LIN {X 0,Y 421.138,Z 564.023,A -85,B 0,C 180,E1 -10017.814,E2 -10017.814} C_VEL
LIN {X 0,Y 421.923,Z 552.011,A -85,B 0,C 180,E1 -10018.748,E2 -10018.748} C_VEL
LIN {X 0,Y 422.666,Z 540.319,A -85,B 0,C 180,E1 -10019.442,E2 -10019.442} C_VEL
LIN {X 0,Y 423.16,Z 527.88,A -85,B 0,C 180,E1 -10019.985,E2 -10019.985} C_VEL
LIN {X 0,Y 423.537,Z 514.922,A -85,B 0,C 180,E1 -10020.346,E2 -10020.346} C_VEL
LIN {X 0,Y 424.553,Z 431.561,A -85,B 0,C 180,E1 -10021.795,E2 -10021.795} C_VEL
LIN {X 0,Y 420.563,Z 412.408,A -85,B 0,C 180,E1 -10022.358,E2 -10022.358} C_VEL
LIN {X 0,Y 420.281,Z 410.463,A -85,B 0,C 180,E1 -10022.492,E2 -10022.492} C_VEL
LIN {X 0,Y 420.893,Z 401.257,A -85,B 0,C 180,E1 -10024.591,E2 -10024.591} C_VEL
LIN {X 0,Y 420.17,Z 396.256,A -85,B 0,C 180,E1 -10025.832,E2 -10025.832} C_VEL
LIN {X 0,Y 418.279,Z 386.932,A -85,B 0,C 180,E1 -10028.302,E2 -10028.302} C_VEL
LIN {X 0,Y 418.263,Z 386.884,A -85,B 0,C 180,E1 -10030.942,E2 -10030.942} C_VEL
LIN {X 0,Y 418.279,Z 386.883,A -85,B 0,C 180,E1 -10033.739,E2 -10033.739} C_VEL
LIN {X 0,Y 418.263,Z 386.884,A -85,B 0,C 180,E1 -10036.456,E2 -10036.456} C_VEL
LIN {X 0,Y 418.262,Z 386.885,A -85,B 0,C 180,E1 -10039.122,E2 -10039.122} C_VEL
LIN {X 0,Y 418.233,Z 386.883,A -85,B 0,C 180,E1 -10042.164,E2 -10042.164} C_VEL
LIN {X 0,Y 418.259,Z 386.876,A -85,B 0,C 180,E1 -10045.419,E2 -10045.419} C_VEL
LIN {X 0,Y 418.217,Z 386.89,A -85,B 0,C 180,E1 -10048.604,E2 -10048.604} C_VEL
LIN {X 0,Y 418.288,Z 386.877,A -85,B 0,C 180,E1 -10051.936,E2 -10051.936} C_VEL
LIN {X 0,Y 418.282,Z 386.882,A -85,B 0,C 180,E1 -10055.162,E2 -10055.162} C_VEL
LIN {X 0,Y 418.247,Z 386.88,A -85,B 0,C 180,E1 -10058.304,E2 -10058.304} C_VEL
LIN {X 0,Y 418.276,Z 386.878,A -85,B 0,C 180,E1 -10061.383,E2 -10061.383} C_VEL
LIN {X 0,Y 418.294,Z 386.879,A -85,B 0,C 180,E1 -10064.406,E2 -10064.406} C_VEL
LIN {X 0,Y 418.361,Z 386.871,A -85,B 0,C 180,E1 -10067.386,E2 -10067.386} C_VEL
LIN {X 0,Y 418.352,Z 386.865,A -85,B 0,C 180,E1 -10070.329,E2 -10070.329} C_VEL
LIN {X 0,Y 418.485,Z 386.852,A -85,B 0,C 180,E1 -10073.249,E2 -10073.249} C_VEL
LIN {X 0,Y 418.336,Z 386.875,A -85,B 0,C 180,E1 -10075.182,E2 -10075.182} C_VEL
LIN {X 0,Y 418.538,Z 386.846,A -85,B 0,C 180,E1 -10078.076,E2 -10078.076} C_VEL
LIN {X 0,Y 418.665,Z 386.828,A -85,B 0,C 180,E1 -10080,E2 -10080} C_VEL
LIN {X 0,Y 418.504,Z 386.851,A -85,B 0,C 180,E1 -10082.888,E2 -10082.888} C_VEL
LIN {X 0,Y 418.486,Z 386.859,A -85,B 0,C 180,E1 -10086.751,E2 -10086.751} C_VEL
LIN {X 0,Y 418.352,Z 386.867,A -85,B 0,C 180,E1 -10089.671,E2 -10089.671} C_VEL
LIN {X 0,Y 418.347,Z 386.867,A -85,B 0,C 180,E1 -10093.006,E2 -10093.006} C_VEL
LIN {X 0,Y 418.304,Z 386.88,A -85,B 0,C 180,E1 -10096.736,E2 -10096.736} C_VEL
LIN {X 0,Y 418.263,Z 386.88,A -85,B 0,C 180,E1 -10099.791,E2 -10099.791} C_VEL
LIN {X 0,Y 418.231,Z 386.884,A -85,B 0,C 180,E1 -10102.737,E2 -10102.737} C_VEL
LIN {X 0,Y 418.264,Z 386.88,A -85,B 0,C 180,E1 -10105.905,E2 -10105.905} C_VEL
LIN {X 0,Y 418.258,Z 386.883,A -85,B 0,C 180,E1 -10109.163,E2 -10109.163} C_VEL
LIN {X 0,Y 418.251,Z 386.886,A -85,B 0,C 180,E1 -10112.845,E2 -10112.845} C_VEL
LIN {X 0,Y 418.243,Z 386.888,A -85,B 0,C 180,E1 -10116.24,E2 -10116.24} C_VEL
LIN {X 0,Y 418.261,Z 386.881,A -85,B 0,C 180,E1 -10119.681,E2 -10119.681} C_VEL
LIN {X 0,Y 418.28,Z 386.87,A -85,B 0,C 180,E1 -10122.33,E2 -10122.33} C_VEL
LIN {X 0,Y 418.251,Z 386.88,A -85,B 0,C 180,E1 -10125.112,E2 -10125.112} C_VEL
LIN {X 0,Y 418.239,Z 386.884,A -85,B 0,C 180,E1 -10127.768,E2 -10127.768} C_VEL
LIN {X 0,Y 418.254,Z 386.881,A -85,B 0,C 180,E1 -10130.619,E2 -10130.619} C_VEL
LIN {X 0,Y 418.244,Z 386.881,A -85,B 0,C 180,E1 -10133.977,E2 -10133.977} C_VEL
LIN {X 0,Y 418.256,Z 386.886,A -85,B 0,C 180,E1 -10137.157,E2 -10137.157} C_VEL
LIN {X 0,Y 418.268,Z 386.886,A -85,B 0,C 180,E1 -10140.896,E2 -10140.896} C_VEL
LIN {X 0,Y 418.343,Z 386.992,A -85,B 0,C 180,E1 -10142.829,E2 -10142.829} C_VEL
LIN {X 0,Y 420.436,Z 396.948,A -85,B 0,C 180,E1 -10145.299,E2 -10145.299} C_VEL
LIN {X 0,Y 421.424,Z 403.012,A -85,B 0,C 180,E1 -10146.715,E2 -10146.715} C_VEL
LIN {X 0,Y 420.312,Z 418.167,A -85,B 0,C 180,E1 -10149.954,E2 -10149.954} C_VEL
LIN {X 0,Y 420.149,Z 421.353,A -85,B 0,C 180,E1 -10150.594,E2 -10150.594} C_VEL
LIN {X 0,Y 421.621,Z 428.874,A -85,B 0,C 180,E1 -10150.85,E2 -10150.85} C_VEL
LIN {X 0,Y 424.489,Z 445.436,A -85,B 0,C 180,E1 -10151.3,E2 -10151.3} C_VEL
LIN {X 0,Y 423.431,Z 529.437,A -85,B 0,C 180,E1 -10152.773,E2 -10152.773} C_VEL
LIN {X 0,Y 422.94,Z 543.257,A -85,B 0,C 180,E1 -10153.219,E2 -10153.219} C_VEL
LIN {X 0,Y 422.283,Z 555.661,A -85,B 0,C 180,E1 -10153.814,E2 -10153.814} C_VEL
LIN {X 0,Y 421.5,Z 566.743,A -85,B 0,C 180,E1 -10154.528,E2 -10154.528} C_VEL
LIN {X 0,Y 420.716,Z 578.277,A -85,B 0,C 180,E1 -10155.489,E2 -10155.489} C_VEL
LIN {X 0,Y 419.929,Z 588.676,A -85,B 0,C 180,E1 -10156.573,E2 -10156.573} C_VEL
LIN {X 0,Y 419.309,Z 597.186,A -85,B 0,C 180,E1 -10157.661,E2 -10157.661} C_VEL
LIN {X 0,Y 418.575,Z 605.051,A -85,B 0,C 180,E1 -10158.867,E2 -10158.867} C_VEL
LIN {X 0,Y 418.026,Z 612.748,A -85,B 0,C 180,E1 -10160.322,E2 -10160.322} C_VEL
LIN {X 0,Y 417.549,Z 618.934,A -85,B 0,C 180,E1 -10161.775,E2 -10161.775} C_VEL
LIN {X 0,Y 417.27,Z 623.86,A -85,B 0,C 180,E1 -10163.229,E2 -10163.229} C_VEL
LIN {X 0,Y 417.161,Z 627.67,A -85,B 0,C 180,E1 -10164.684,E2 -10164.684} C_VEL
LIN {X 0,Y 417.001,Z 630.466,A -85,B 0,C 180,E1 -10166.135,E2 -10166.135} C_VEL
LIN {X 0,Y 417.03,Z 632.726,A -85,B 0,C 180,E1 -10168.069,E2 -10168.069} C_VEL
LIN {X 0,Y 416.992,Z 633.268,A -85,B 0,C 180,E1 -10169.035,E2 -10169.035} C_VEL
LIN {X 0,Y 416.982,Z 633.379,A -85,B 0,C 180,E1 -10170,E2 -10170} C_VEL
LIN {X 0,Y 417.03,Z 632.435,A -85,B 0,C 180,E1 -10171.932,E2 -10171.932} C_VEL
LIN {X 0,Y 416.984,Z 631.378,A -85,B 0,C 180,E1 -10172.898,E2 -10172.898} C_VEL
LIN {X 0,Y 417,Z 629.867,A -85,B 0,C 180,E1 -10173.866,E2 -10173.866} C_VEL
LIN {X 0,Y 417.141,Z 626.813,A -85,B 0,C 180,E1 -10175.317,E2 -10175.317} C_VEL
LIN {X 0,Y 417.244,Z 622.691,A -85,B 0,C 180,E1 -10176.771,E2 -10176.771} C_VEL
LIN {X 0,Y 417.566,Z 616.376,A -85,B 0,C 180,E1 -10178.469,E2 -10178.469} C_VEL
LIN {X 0,Y 417.985,Z 609.49,A -85,B 0,C 180,E1 -10179.924,E2 -10179.924} C_VEL
LIN {X 0,Y 418.42,Z 602.45,A -85,B 0,C 180,E1 -10181.137,E2 -10181.137} C_VEL
LIN {X 0,Y 419.055,Z 593.964,A -85,B 0,C 180,E1 -10182.347,E2 -10182.347} C_VEL
LIN {X 0,Y 419.747,Z 583.455,A -85,B 0,C 180,E1 -10183.557,E2 -10183.557} C_VEL
LIN {X 0,Y 420.461,Z 571.606,A -85,B 0,C 180,E1 -10184.644,E2 -10184.644} C_VEL
LIN {X 0,Y 421.178,Z 559.68,A -85,B 0,C 180,E1 -10185.485,E2 -10185.485} C_VEL
LIN {X 0,Y 421.793,Z 547.253,A -85,B 0,C 180,E1 -10186.144,E2 -10186.144} C_VEL
LIN {X 0,Y 422.289,Z 534.454,A -85,B 0,C 180,E1 -10186.621,E2 -10186.621} C_VEL
LIN {X 0,Y 422.514,Z 520.889,A -85,B 0,C 180,E1 -10186.923,E2 -10186.923} C_VEL
LIN {X 0,Y 423.276,Z 444.977,A -85,B 0,C 180,E1 -10188.213,E2 -10188.213} C_VEL
LIN {X 0,Y 419.583,Z 421.755,A -85,B 0,C 180,E1 -10188.779,E2 -10188.779} C_VEL
LIN {X 0,Y 419.773,Z 417.624,A -85,B 0,C 180,E1 -10189.563,E2 -10189.563} C_VEL
LIN {X 0,Y 420.813,Z 401.434,A -85,B 0,C 180,E1 -10192.923,E2 -10192.923} C_VEL
LIN {X 0,Y 419.777,Z 394.378,A -85,B 0,C 180,E1 -10194.479,E2 -10194.479} C_VEL
LIN {X 0,Y 418.35,Z 386.974,A -85,B 0,C 180,E1 -10196.2,E2 -10196.2} C_VEL
LIN {X 0,Y 418.266,Z 386.886,A -85,B 0,C 180,E1 -10199.161,E2 -10199.161} C_VEL
LIN {X 0,Y 418.258,Z 386.882,A -85,B 0,C 180,E1 -10202.844,E2 -10202.844} C_VEL
LIN {X 0,Y 418.249,Z 386.884,A -85,B 0,C 180,E1 -10206.238,E2 -10206.238} C_VEL
LIN {X 0,Y 418.255,Z 386.886,A -85,B 0,C 180,E1 -10209.681,E2 -10209.681} C_VEL
LIN {X 0,Y 418.231,Z 386.886,A -85,B 0,C 180,E1 -10212.321,E2 -10212.321} C_VEL
LIN {X 0,Y 418.26,Z 386.885,A -85,B 0,C 180,E1 -10215.112,E2 -10215.112} C_VEL
LIN {X 0,Y 418.291,Z 386.881,A -85,B 0,C 180,E1 -10217.773,E2 -10217.773} C_VEL
LIN {X 0,Y 418.264,Z 386.885,A -85,B 0,C 180,E1 -10221.559,E2 -10221.559} C_VEL
LIN {X 0,Y 418.256,Z 386.887,A -85,B 0,C 180,E1 -10225.159,E2 -10225.159} C_VEL
LIN {X 0,Y 418.242,Z 386.888,A -85,B 0,C 180,E1 -10227.471,E2 -10227.471} C_VEL
LIN {X 0,Y 418.265,Z 386.884,A -85,B 0,C 180,E1 -10230.895,E2 -10230.895} C_VEL
LIN {X 0,Y 418.267,Z 386.883,A -85,B 0,C 180,E1 -10234.096,E2 -10234.096} C_VEL
LIN {X 0,Y 418.227,Z 386.891,A -85,B 0,C 180,E1 -10237.263,E2 -10237.263} C_VEL
LIN {X 0,Y 418.278,Z 386.88,A -85,B 0,C 180,E1 -10240.364,E2 -10240.364} C_VEL
LIN {X 0,Y 418.312,Z 386.879,A -85,B 0,C 180,E1 -10243.404,E2 -10243.404} C_VEL
LIN {X 0,Y 418.341,Z 386.876,A -85,B 0,C 180,E1 -10246.999,E2 -10246.999} C_VEL
LIN {X 0,Y 418.335,Z 386.874,A -85,B 0,C 180,E1 -10250.328,E2 -10250.328} C_VEL
LIN {X 0,Y 418.487,Z 386.858,A -85,B 0,C 180,E1 -10253.249,E2 -10253.249} C_VEL
LIN {X 0,Y 418.335,Z 386.877,A -85,B 0,C 180,E1 -10255.181,E2 -10255.181} C_VEL
LIN {X 0,Y 418.539,Z 386.849,A -85,B 0,C 180,E1 -10258.075,E2 -10258.075} C_VEL
LIN {X 0,Y 418.666,Z 386.833,A -85,B 0,C 180,E1 -10260,E2 -10260} C_VEL
LIN {X 0,Y 418.505,Z 386.855,A -85,B 0,C 180,E1 -10262.888,E2 -10262.888} C_VEL
LIN {X 0,Y 418.488,Z 386.857,A -85,B 0,C 180,E1 -10266.751,E2 -10266.751} C_VEL
LIN {X 0,Y 418.335,Z 386.876,A -85,B 0,C 180,E1 -10269.671,E2 -10269.671} C_VEL
LIN {X 0,Y 418.34,Z 386.876,A -85,B 0,C 180,E1 -10273.001,E2 -10273.001} C_VEL
LIN {X 0,Y 418.307,Z 386.879,A -85,B 0,C 180,E1 -10276.736,E2 -10276.736} C_VEL
LIN {X 0,Y 418.265,Z 386.884,A -85,B 0,C 180,E1 -10279.79,E2 -10279.79} C_VEL
LIN {X 0,Y 418.233,Z 386.889,A -85,B 0,C 180,E1 -10282.736,E2 -10282.736} C_VEL
LIN {X 0,Y 418.266,Z 386.883,A -85,B 0,C 180,E1 -10285.904,E2 -10285.904} C_VEL
LIN {X 0,Y 418.27,Z 386.884,A -85,B 0,C 180,E1 -10289.162,E2 -10289.162} C_VEL
LIN {X 0,Y 418.254,Z 386.886,A -85,B 0,C 180,E1 -10292.844,E2 -10292.844} C_VEL
LIN {X 0,Y 418.245,Z 386.885,A -85,B 0,C 180,E1 -10296.239,E2 -10296.239} C_VEL
LIN {X 0,Y 418.249,Z 386.885,A -85,B 0,C 180,E1 -10299.682,E2 -10299.682} C_VEL
LIN {X 0,Y 418.229,Z 386.887,A -85,B 0,C 180,E1 -10302.322,E2 -10302.322} C_VEL
LIN {X 0,Y 418.235,Z 386.89,A -85,B 0,C 180,E1 -10305.109,E2 -10305.109} C_VEL
LIN {X 0,Y 418.254,Z 386.884,A -85,B 0,C 180,E1 -10307.769,E2 -10307.769} C_VEL
LIN {X 0,Y 418.266,Z 386.883,A -85,B 0,C 180,E1 -10310.617,E2 -10310.617} C_VEL
LIN {X 0,Y 418.245,Z 386.884,A -85,B 0,C 180,E1 -10313.977,E2 -10313.977} C_VEL
LIN {X 0,Y 418.257,Z 386.888,A -85,B 0,C 180,E1 -10317.156,E2 -10317.156} C_VEL
LIN {X 0,Y 418.268,Z 386.885,A -85,B 0,C 180,E1 -10320.896,E2 -10320.896} C_VEL
LIN {X 0,Y 418.271,Z 386.88,A -85,B 0,C 180,E1 -10324.096,E2 -10324.096} C_VEL
LIN {X 0,Y 418.239,Z 386.888,A -85,B 0,C 180,E1 -10327.264,E2 -10327.264} C_VEL
LIN {X 0,Y 418.284,Z 386.879,A -85,B 0,C 180,E1 -10330.364,E2 -10330.364} C_VEL
LIN {X 0,Y 418.318,Z 386.876,A -85,B 0,C 180,E1 -10333.405,E2 -10333.405} C_VEL
LIN {X 0,Y 418.348,Z 386.877,A -85,B 0,C 180,E1 -10336.999,E2 -10336.999} C_VEL
LIN {X 0,Y 418.318,Z 386.913,A -85,B 0,C 180,E1 -10338.737,E2 -10338.737} C_VEL
LIN {X 0,Y 419.362,Z 392.298,A -85,B 0,C 180,E1 -10340.109,E2 -10340.109} C_VEL
LIN {X 0,Y 420.285,Z 398.53,A -85,B 0,C 180,E1 -10341.586,E2 -10341.586} C_VEL
LIN {X 0,Y 419.795,Z 404.966,A -85,B 0,C 180,E1 -10343.028,E2 -10343.028} C_VEL
LIN {X 0,Y 419.5,Z 409.848,A -85,B 0,C 180,E1 -10344.11,E2 -10344.11} C_VEL
LIN {X 0,Y 419.508,Z 410.969,A -85,B 0,C 180,E1 -10344.274,E2 -10344.274} C_VEL
LIN {X 0,Y 422.211,Z 425.053,A -85,B 0,C 180,E1 -10344.648,E2 -10344.648} C_VEL
LIN {X 0,Y 423.411,Z 432.135,A -85,B 0,C 180,E1 -10344.818,E2 -10344.818} C_VEL
LIN {X 0,Y 422.442,Z 518.153,A -85,B 0,C 180,E1 -10346.304,E2 -10346.304} C_VEL
LIN {X 0,Y 422.1,Z 529.926,A -85,B 0,C 180,E1 -10346.669,E2 -10346.669} C_VEL
LIN {X 0,Y 420.303,Z 537.386,A -85,B 0,C 180,E1 -10346.935,E2 -10346.935} C_VEL
LIN {X 0,Y 417.529,Z 544.56,A -85,B 0,C 180,E1 -10347.223,E2 -10347.223} C_VEL
LIN {X 0,Y 414.552,Z 553.329,A -85,B 0,C 180,E1 -10347.702,E2 -10347.702} C_VEL
LIN {X 0,Y 413.762,Z 558.483,A -85,B 0,C 180,E1 -10348.072,E2 -10348.072} C_VEL
LIN {X 0,Y 413.074,Z 569.244,A -85,B 0,C 180,E1 -10349.025,E2 -10349.025} C_VEL
LIN {X 0,Y 412.365,Z 578.193,A -85,B 0,C 180,E1 -10350,E2 -10350} C_VEL
LIN {X 0,Y 411.779,Z 587.346,A -85,B 0,C 180,E1 -10351.222,E2 -10351.222} C_VEL
LIN {X 0,Y 411.1,Z 596.284,A -85,B 0,C 180,E1 -10352.694,E2 -10352.694} C_VEL
LIN {X 0,Y 410.64,Z 603.483,A -85,B 0,C 180,E1 -10354.171,E2 -10354.171} C_VEL
LIN {X 0,Y 410.383,Z 608.342,A -85,B 0,C 180,E1 -10355.404,E2 -10355.404} C_VEL
LIN {X 0,Y 410.176,Z 613.073,A -85,B 0,C 180,E1 -10356.888,E2 -10356.888} C_VEL
LIN {X 0,Y 409.998,Z 616.699,A -85,B 0,C 180,E1 -10358.378,E2 -10358.378} C_VEL
LIN {X 0,Y 409.821,Z 619.308,A -85,B 0,C 180,E1 -10359.874,E2 -10359.874} C_VEL
LIN {X 0,Y 409.852,Z 620.528,A -85,B 0,C 180,E1 -10360.872,E2 -10360.872} C_VEL
LIN {X 0,Y 409.883,Z 621.466,A -85,B 0,C 180,E1 -10362.22,E2 -10362.22} C_VEL
LIN {X 0,Y 409.755,Z 621.629,A -85,B 0,C 180,E1 -10363.893,E2 -10363.893} C_VEL
LIN {X 0,Y 409.778,Z 621.181,A -85,B 0,C 180,E1 -10364.907,E2 -10364.907} C_VEL
LIN {X 0,Y 409.86,Z 619.948,A -85,B 0,C 180,E1 -10366.209,E2 -10366.209} C_VEL
LIN {X 0,Y 410.018,Z 617.188,A -85,B 0,C 180,E1 -10367.97,E2 -10367.97} C_VEL
LIN {X 0,Y 410.269,Z 613.417,A -85,B 0,C 180,E1 -10369.582,E2 -10369.582} C_VEL
LIN {X 0,Y 410.586,Z 608.813,A -85,B 0,C 180,E1 -10371.066,E2 -10371.066} C_VEL
LIN {X 0,Y 411.167,Z 601.801,A -85,B 0,C 180,E1 -10372.81,E2 -10372.81} C_VEL
LIN {X 0,Y 411.73,Z 594.877,A -85,B 0,C 180,E1 -10374.183,E2 -10374.183} C_VEL
LIN {X 0,Y 412.462,Z 586.649,A -85,B 0,C 180,E1 -10375.516,E2 -10375.516} C_VEL
LIN {X 0,Y 413.27,Z 576.951,A -85,B 0,C 180,E1 -10376.785,E2 -10376.785} C_VEL
LIN {X 0,Y 414.145,Z 566.829,A -85,B 0,C 180,E1 -10377.854,E2 -10377.854} C_VEL
LIN {X 0,Y 414.981,Z 554.936,A -85,B 0,C 180,E1 -10378.859,E2 -10378.859} C_VEL
LIN {X 0,Y 415.794,Z 542.865,A -85,B 0,C 180,E1 -10379.629,E2 -10379.629} C_VEL
LIN {X 0,Y 416.433,Z 529.777,A -85,B 0,C 180,E1 -10380.242,E2 -10380.242} C_VEL
LIN {X 0,Y 416.877,Z 517.663,A -85,B 0,C 180,E1 -10380.618,E2 -10380.618} C_VEL
LIN {X 0,Y 417.981,Z 432.664,A -85,B 0,C 180,E1 -10382.127,E2 -10382.127} C_VEL
LIN {X 0,Y 413.773,Z 412.697,A -85,B 0,C 180,E1 -10382.735,E2 -10382.735} C_VEL
LIN {X 0,Y 413.455,Z 410.579,A -85,B 0,C 180,E1 -10382.875,E2 -10382.875} C_VEL
LIN {X 0,Y 413.984,Z 402.873,A -85,B 0,C 180,E1 -10384.659,E2 -10384.659} C_VEL
LIN {X 0,Y 413.541,Z 399.14,A -85,B 0,C 180,E1 -10385.594,E2 -10385.594} C_VEL
LIN {X 0,Y 411.249,Z 387.872,A -85,B 0,C 180,E1 -10388.594,E2 -10388.594} C_VEL
LIN {X 0,Y 411.217,Z 387.764,A -85,B 0,C 180,E1 -10391.799,E2 -10391.799} C_VEL
LIN {X 0,Y 411.232,Z 387.761,A -85,B 0,C 180,E1 -10394.481,E2 -10394.481} C_VEL
LIN {X 0,Y 411.224,Z 387.758,A -85,B 0,C 180,E1 -10397.296,E2 -10397.296} C_VEL
LIN {X 0,Y 411.226,Z 387.757,A -85,B 0,C 180,E1 -10400.777,E2 -10400.777} C_VEL
LIN {X 0,Y 411.194,Z 387.762,A -85,B 0,C 180,E1 -10404.471,E2 -10404.471} C_VEL
LIN {X 0,Y 411.166,Z 387.766,A -85,B 0,C 180,E1 -10408.003,E2 -10408.003} C_VEL
LIN {X 0,Y 411.217,Z 387.757,A -85,B 0,C 180,E1 -10411.41,E2 -10411.41} C_VEL
LIN {X 0,Y 411.229,Z 387.759,A -85,B 0,C 180,E1 -10414.706,E2 -10414.706} C_VEL
LIN {X 0,Y 411.222,Z 387.754,A -85,B 0,C 180,E1 -10417.914,E2 -10417.914} C_VEL
LIN {X 0,Y 411.228,Z 387.758,A -85,B 0,C 180,E1 -10421.052,E2 -10421.052} C_VEL
LIN {X 0,Y 411.246,Z 387.756,A -85,B 0,C 180,E1 -10424.131,E2 -10424.131} C_VEL
LIN {X 0,Y 411.306,Z 387.752,A -85,B 0,C 180,E1 -10427.166,E2 -10427.166} C_VEL
LIN {X 0,Y 411.3,Z 387.742,A -85,B 0,C 180,E1 -10430.161,E2 -10430.161} C_VEL
LIN {X 0,Y 411.452,Z 387.729,A -85,B 0,C 180,E1 -10433.133,E2 -10433.133} C_VEL
LIN {X 0,Y 411.307,Z 387.749,A -85,B 0,C 180,E1 -10435.099,E2 -10435.099} C_VEL
LIN {X 0,Y 411.507,Z 387.721,A -85,B 0,C 180,E1 -10438.043,E2 -10438.043} C_VEL
LIN {X 0,Y 411.635,Z 387.703,A -85,B 0,C 180,E1 -10440,E2 -10440} C_VEL
LIN {X 0,Y 411.459,Z 387.727,A -85,B 0,C 180,E1 -10442.937,E2 -10442.937} C_VEL
LIN {X 0,Y 411.452,Z 387.733,A -85,B 0,C 180,E1 -10446.867,E2 -10446.867} C_VEL
LIN {X 0,Y 411.3,Z 387.746,A -85,B 0,C 180,E1 -10449.839,E2 -10449.839} C_VEL
LIN {X 0,Y 411.305,Z 387.743,A -85,B 0,C 180,E1 -10453.109,E2 -10453.109} C_VEL
LIN {X 0,Y 411.249,Z 387.756,A -85,B 0,C 180,E1 -10456.889,E2 -10456.889} C_VEL
LIN {X 0,Y 411.223,Z 387.758,A -85,B 0,C 180,E1 -10459.987,E2 -10459.987} C_VEL
LIN {X 0,Y 411.196,Z 387.762,A -85,B 0,C 180,E1 -10463.148,E2 -10463.148} C_VEL
LIN {X 0,Y 411.231,Z 387.758,A -85,B 0,C 180,E1 -10466.382,E2 -10466.382} C_VEL
LIN {X 0,Y 411.193,Z 387.761,A -85,B 0,C 180,E1 -10469.713,E2 -10469.713} C_VEL
LIN {X 0,Y 411.2,Z 387.761,A -85,B 0,C 180,E1 -10473.157,E2 -10473.157} C_VEL
LIN {X 0,Y 411.19,Z 387.766,A -85,B 0,C 180,E1 -10476.554,E2 -10476.554} C_VEL
LIN {X 0,Y 411.223,Z 387.758,A -85,B 0,C 180,E1 -10479.731,E2 -10479.731} C_VEL
LIN {X 0,Y 411.218,Z 387.761,A -85,B 0,C 180,E1 -10483.128,E2 -10483.128} C_VEL
LIN {X 0,Y 411.173,Z 387.76,A -85,B 0,C 180,E1 -10485.881,E2 -10485.881} C_VEL
LIN {X 0,Y 411.202,Z 387.759,A -85,B 0,C 180,E1 -10489.5,E2 -10489.5} C_VEL
LIN {X 0,Y 411.198,Z 387.766,A -85,B 0,C 180,E1 -10492.028,E2 -10492.028} C_VEL
LIN {X 0,Y 411.205,Z 387.762,A -85,B 0,C 180,E1 -10495.667,E2 -10495.667} C_VEL
LIN {X 0,Y 411.188,Z 387.767,A -85,B 0,C 180,E1 -10499.153,E2 -10499.153} C_VEL
LIN {X 0,Y 411.324,Z 387.969,A -85,B 0,C 180,E1 -10502.528,E2 -10502.528} C_VEL
LIN {X 0,Y 413.717,Z 399.466,A -85,B 0,C 180,E1 -10505.406,E2 -10505.406} C_VEL
LIN {X 0,Y 414.504,Z 404.905,A -85,B 0,C 180,E1 -10506.691,E2 -10506.691} C_VEL
LIN {X 0,Y 413.277,Z 421.152,A -85,B 0,C 180,E1 -10510.19,E2 -10510.19} C_VEL
LIN {X 0,Y 414.015,Z 425.012,A -85,B 0,C 180,E1 -10510.358,E2 -10510.358} C_VEL
LIN {X 0,Y 417.605,Z 444.687,A -85,B 0,C 180,E1 -10510.922,E2 -10510.922} C_VEL
LIN {X 0,Y 417.86,Z 448.094,A -85,B 0,C 180,E1 -10510.997,E2 -10510.997} C_VEL
LIN {X 0,Y 416.796,Z 528.713,A -85,B 0,C 180,E1 -10512.427,E2 -10512.427} C_VEL
LIN {X 0,Y 416.268,Z 541.999,A -85,B 0,C 180,E1 -10512.847,E2 -10512.847} C_VEL
LIN {X 0,Y 415.611,Z 554.148,A -85,B 0,C 180,E1 -10513.42,E2 -10513.42} C_VEL
LIN {X 0,Y 414.869,Z 565.595,A -85,B 0,C 180,E1 -10514.148,E2 -10514.148} C_VEL
LIN {X 0,Y 413.95,Z 577.353,A -85,B 0,C 180,E1 -10515.121,E2 -10515.121} C_VEL
LIN {X 0,Y 413.099,Z 587.882,A -85,B 0,C 180,E1 -10516.221,E2 -10516.221} C_VEL
LIN {X 0,Y 412.386,Z 597.385,A -85,B 0,C 180,E1 -10517.451,E2 -10517.451} C_VEL
LIN {X 0,Y 411.58,Z 605.19,A -85,B 0,C 180,E1 -10518.676,E2 -10518.676} C_VEL
LIN {X 0,Y 411.011,Z 612.823,A -85,B 0,C 180,E1 -10520.155,E2 -10520.155} C_VEL
LIN {X 0,Y 410.523,Z 618.975,A -85,B 0,C 180,E1 -10521.633,E2 -10521.633} C_VEL
LIN {X 0,Y 410.196,Z 623.871,A -85,B 0,C 180,E1 -10523.112,E2 -10523.112} C_VEL
LIN {X 0,Y 410.079,Z 627.653,A -85,B 0,C 180,E1 -10524.592,E2 -10524.592} C_VEL
LIN {X 0,Y 409.923,Z 630.423,A -85,B 0,C 180,E1 -10526.068,E2 -10526.068} C_VEL
LIN {X 0,Y 409.926,Z 632.657,A -85,B 0,C 180,E1 -10528.035,E2 -10528.035} C_VEL
LIN {X 0,Y 409.918,Z 633.179,A -85,B 0,C 180,E1 -10529.018,E2 -10529.018} C_VEL
LIN {X 0,Y 409.918,Z 632.98,A -85,B 0,C 180,E1 -10530.983,E2 -10530.983} C_VEL
LIN {X 0,Y 409.926,Z 632.303,A -85,B 0,C 180,E1 -10531.965,E2 -10531.965} C_VEL
LIN {X 0,Y 409.883,Z 631.226,A -85,B 0,C 180,E1 -10532.949,E2 -10532.949} C_VEL
LIN {X 0,Y 409.92,Z 629.695,A -85,B 0,C 180,E1 -10533.933,E2 -10533.933} C_VEL
LIN {X 0,Y 410.038,Z 626.612,A -85,B 0,C 180,E1 -10535.409,E2 -10535.409} C_VEL
LIN {X 0,Y 410.181,Z 622.461,A -85,B 0,C 180,E1 -10536.889,E2 -10536.889} C_VEL
LIN {X 0,Y 410.53,Z 616.113,A -85,B 0,C 180,E1 -10538.615,E2 -10538.615} C_VEL
LIN {X 0,Y 410.96,Z 609.189,A -85,B 0,C 180,E1 -10540.096,E2 -10540.096} C_VEL
LIN {X 0,Y 411.42,Z 602.108,A -85,B 0,C 180,E1 -10541.329,E2 -10541.329} C_VEL
LIN {X 0,Y 412.081,Z 593.556,A -85,B 0,C 180,E1 -10542.559,E2 -10542.559} C_VEL
LIN {X 0,Y 412.797,Z 582.971,A -85,B 0,C 180,E1 -10543.789,E2 -10543.789} C_VEL
LIN {X 0,Y 413.454,Z 572.476,A -85,B 0,C 180,E1 -10544.772,E2 -10544.772} C_VEL
LIN {X 0,Y 414.17,Z 560.91,A -85,B 0,C 180,E1 -10545.627,E2 -10545.627} C_VEL
LIN {X 0,Y 414.804,Z 548.892,A -85,B 0,C 180,E1 -10546.297,E2 -10546.297} C_VEL
LIN {X 0,Y 415.354,Z 535.884,A -85,B 0,C 180,E1 -10546.812,E2 -10546.812} C_VEL
LIN {X 0,Y 415.618,Z 523.662,A -85,B 0,C 180,E1 -10547.118,E2 -10547.118} C_VEL
LIN {X 0,Y 416.464,Z 446.016,A -85,B 0,C 180,E1 -10548.457,E2 -10548.457} C_VEL
LIN {X 0,Y 412.612,Z 421.485,A -85,B 0,C 180,E1 -10549.076,E2 -10549.076} C_VEL
LIN {X 0,Y 413.551,Z 406.335,A -85,B 0,C 180,E1 -10552.217,E2 -10552.217} C_VEL
LIN {X 0,Y 413.777,Z 401.214,A -85,B 0,C 180,E1 -10553.309,E2 -10553.309} C_VEL
LIN {X 0,Y 411.517,Z 389.025,A -85,B 0,C 180,E1 -10556.088,E2 -10556.088} C_VEL
LIN {X 0,Y 411.314,Z 387.774,A -85,B 0,C 180,E1 -10556.477,E2 -10556.477} C_VEL
LIN {X 0,Y 411.201,Z 387.765,A -85,B 0,C 180,E1 -10559.712,E2 -10559.712} C_VEL
LIN {X 0,Y 411.207,Z 387.762,A -85,B 0,C 180,E1 -10563.155,E2 -10563.155} C_VEL
LIN {X 0,Y 411.195,Z 387.761,A -85,B 0,C 180,E1 -10566.553,E2 -10566.553} C_VEL
LIN {X 0,Y 411.218,Z 387.762,A -85,B 0,C 180,E1 -10569.728,E2 -10569.728} C_VEL
LIN {X 0,Y 411.177,Z 387.767,A -85,B 0,C 180,E1 -10573.132,E2 -10573.132} C_VEL
LIN {X 0,Y 411.226,Z 387.76,A -85,B 0,C 180,E1 -10575.872,E2 -10575.872} C_VEL
LIN {X 0,Y 411.208,Z 387.761,A -85,B 0,C 180,E1 -10578.764,E2 -10578.764} C_VEL
LIN {X 0,Y 411.203,Z 387.763,A -85,B 0,C 180,E1 -10582.027,E2 -10582.027} C_VEL
LIN {X 0,Y 411.203,Z 387.764,A -85,B 0,C 180,E1 -10585.666,E2 -10585.666} C_VEL
LIN {X 0,Y 411.186,Z 387.767,A -85,B 0,C 180,E1 -10589.152,E2 -10589.152} C_VEL
LIN {X 0,Y 411.255,Z 387.755,A -85,B 0,C 180,E1 -10592.522,E2 -10592.522} C_VEL
LIN {X 0,Y 411.216,Z 387.762,A -85,B 0,C 180,E1 -10595.784,E2 -10595.784} C_VEL
LIN {X 0,Y 411.191,Z 387.766,A -85,B 0,C 180,E1 -10598.965,E2 -10598.965} C_VEL
LIN {X 0,Y 411.248,Z 387.757,A -85,B 0,C 180,E1 -10602.085,E2 -10602.085} C_VEL
LIN {X 0,Y 411.254,Z 387.76,A -85,B 0,C 180,E1 -10605.147,E2 -10605.147} C_VEL
LIN {X 0,Y 411.278,Z 387.753,A -85,B 0,C 180,E1 -10608.167,E2 -10608.167} C_VEL
LIN {X 0,Y 411.435,Z 387.733,A -85,B 0,C 180,E1 -10612.189,E2 -10612.189} C_VEL
LIN {X 0,Y 411.469,Z 387.729,A -85,B 0,C 180,E1 -10614.118,E2 -10614.118} C_VEL
LIN {X 0,Y 411.508,Z 387.724,A -85,B 0,C 180,E1 -10618.042,E2 -10618.042} C_VEL
LIN {X 0,Y 411.636,Z 387.709,A -85,B 0,C 180,E1 -10620,E2 -10620} C_VEL
LIN {X 0,Y 411.461,Z 387.733,A -85,B 0,C 180,E1 -10622.937,E2 -10622.937} C_VEL
LIN {X 0,Y 411.455,Z 387.733,A -85,B 0,C 180,E1 -10626.867,E2 -10626.867} C_VEL
LIN {X 0,Y 411.287,Z 387.753,A -85,B 0,C 180,E1 -10629.839,E2 -10629.839} C_VEL
LIN {X 0,Y 411.3,Z 387.753,A -85,B 0,C 180,E1 -10633.104,E2 -10633.104} C_VEL
LIN {X 0,Y 411.252,Z 387.759,A -85,B 0,C 180,E1 -10636.889,E2 -10636.889} C_VEL
LIN {X 0,Y 411.225,Z 387.759,A -85,B 0,C 180,E1 -10639.987,E2 -10639.987} C_VEL
LIN {X 0,Y 411.198,Z 387.765,A -85,B 0,C 180,E1 -10643.148,E2 -10643.148} C_VEL
LIN {X 0,Y 411.233,Z 387.758,A -85,B 0,C 180,E1 -10646.381,E2 -10646.381} C_VEL
LIN {X 0,Y 411.207,Z 387.763,A -85,B 0,C 180,E1 -10649.712,E2 -10649.712} C_VEL
LIN {X 0,Y 411.202,Z 387.765,A -85,B 0,C 180,E1 -10653.156,E2 -10653.156} C_VEL
LIN {X 0,Y 411.192,Z 387.764,A -85,B 0,C 180,E1 -10656.553,E2 -10656.553} C_VEL
LIN {X 0,Y 411.212,Z 387.761,A -85,B 0,C 180,E1 -10659.729,E2 -10659.729} C_VEL
LIN {X 0,Y 411.175,Z 387.769,A -85,B 0,C 180,E1 -10663.133,E2 -10663.133} C_VEL
LIN {X 0,Y 411.166,Z 387.766,A -85,B 0,C 180,E1 -10665.881,E2 -10665.881} C_VEL
LIN {X 0,Y 411.198,Z 387.764,A -85,B 0,C 180,E1 -10668.766,E2 -10668.766} C_VEL
LIN {X 0,Y 411.203,Z 387.761,A -85,B 0,C 180,E1 -10672.028,E2 -10672.028} C_VEL
LIN {X 0,Y 411.205,Z 387.762,A -85,B 0,C 180,E1 -10675.667,E2 -10675.667} C_VEL
LIN {X 0,Y 411.189,Z 387.768,A -85,B 0,C 180,E1 -10679.153,E2 -10679.153} C_VEL
LIN {X 0,Y 411.259,Z 387.756,A -85,B 0,C 180,E1 -10682.523,E2 -10682.523} C_VEL
LIN {X 0,Y 411.227,Z 387.758,A -85,B 0,C 180,E1 -10685.785,E2 -10685.785} C_VEL
LIN {X 0,Y 411.197,Z 387.767,A -85,B 0,C 180,E1 -10688.966,E2 -10688.966} C_VEL
LIN {X 0,Y 411.254,Z 387.754,A -85,B 0,C 180,E1 -10692.085,E2 -10692.085} C_VEL
LIN {X 0,Y 411.262,Z 387.759,A -85,B 0,C 180,E1 -10695.147,E2 -10695.147} C_VEL
LIN {X 0,Y 411.299,Z 387.754,A -85,B 0,C 180,E1 -10698.418,E2 -10698.418} C_VEL
LIN {X 0,Y 411.346,Z 388.079,A -85,B 0,C 180,E1 -10698.669,E2 -10698.669} C_VEL
LIN {X 0,Y 413.232,Z 398.371,A -85,B 0,C 180,E1 -10701.195,E2 -10701.195} C_VEL
LIN {X 0,Y 412.812,Z 405.854,A -85,B 0,C 180,E1 -10702.91,E2 -10702.91} C_VEL
LIN {X 0,Y 412.541,Z 410.618,A -85,B 0,C 180,E1 -10703.949,E2 -10703.949} C_VEL
LIN {X 0,Y 412.899,Z 413.107,A -85,B 0,C 180,E1 -10704.071,E2 -10704.071} C_VEL
LIN {X 0,Y 416.584,Z 433.301,A -85,B 0,C 180,E1 -10704.573,E2 -10704.573} C_VEL
LIN {X 0,Y 415.588,Z 517.953,A -85,B 0,C 180,E1 -10706.054,E2 -10706.054} C_VEL
LIN {X 0,Y 415.171,Z 530.499,A -85,B 0,C 180,E1 -10706.451,E2 -10706.451} C_VEL
LIN {X 0,Y 414.599,Z 543.854,A -85,B 0,C 180,E1 -10707.085,E2 -10707.085} C_VEL
LIN {X 0,Y 413.997,Z 555.078,A -85,B 0,C 180,E1 -10707.811,E2 -10707.811} C_VEL
LIN {X 0,Y 413.762,Z 558.483,A -85,B 0,C 180,E1 -10708.072,E2 -10708.072} C_VEL
LIN {X 0,Y 412.834,Z 563.554,A -85,B 0,C 180,E1 -10708.473,E2 -10708.473} C_VEL
LIN {X 0,Y 409.42,Z 571.503,A -85,B 0,C 180,E1 -10709.154,E2 -10709.154} C_VEL
LIN {X 0,Y 405.985,Z 579.039,A -85,B 0,C 180,E1 -10709.931,E2 -10709.931} C_VEL
LIN {X 0,Y 405.034,Z 583.369,A -85,B 0,C 180,E1 -10710.478,E2 -10710.478} C_VEL
LIN {X 0,Y 404.411,Z 591.763,A -85,B 0,C 180,E1 -10711.742,E2 -10711.742} C_VEL
LIN {X 0,Y 403.844,Z 599.854,A -85,B 0,C 180,E1 -10713.242,E2 -10713.242} C_VEL
LIN {X 0,Y 403.366,Z 605.373,A -85,B 0,C 180,E1 -10714.497,E2 -10714.497} C_VEL
LIN {X 0,Y 403.196,Z 610.746,A -85,B 0,C 180,E1 -10716.003,E2 -10716.003} C_VEL
LIN {X 0,Y 403.017,Z 614.958,A -85,B 0,C 180,E1 -10717.515,E2 -10717.515} C_VEL
LIN {X 0,Y 402.813,Z 618.113,A -85,B 0,C 180,E1 -10719.034,E2 -10719.034} C_VEL
LIN {X 0,Y 402.729,Z 619.683,A -85,B 0,C 180,E1 -10720.05,E2 -10720.05} C_VEL
LIN {X 0,Y 402.747,Z 620.793,A -85,B 0,C 180,E1 -10721.066,E2 -10721.066} C_VEL
LIN {X 0,Y 402.786,Z 621.583,A -85,B 0,C 180,E1 -10722.281,E2 -10722.281} C_VEL
LIN {X 0,Y 402.667,Z 621.691,A -85,B 0,C 180,E1 -10724.143,E2 -10724.143} C_VEL
LIN {X 0,Y 402.706,Z 621.13,A -85,B 0,C 180,E1 -10725.175,E2 -10725.175} C_VEL
LIN {X 0,Y 402.767,Z 620.036,A -85,B 0,C 180,E1 -10726.319,E2 -10726.319} C_VEL
LIN {X 0,Y 402.849,Z 618.767,A -85,B 0,C 180,E1 -10727.252,E2 -10727.252} C_VEL
LIN {X 0,Y 403.066,Z 615.788,A -85,B 0,C 180,E1 -10728.818,E2 -10728.818} C_VEL
LIN {X 0,Y 403.348,Z 611.68,A -85,B 0,C 180,E1 -10730.394,E2 -10730.394} C_VEL
LIN {X 0,Y 403.872,Z 605.239,A -85,B 0,C 180,E1 -10732.239,E2 -10732.239} C_VEL
LIN {X 0,Y 404.513,Z 598.133,A -85,B 0,C 180,E1 -10733.824,E2 -10733.824} C_VEL
LIN {X 0,Y 405.191,Z 590.799,A -85,B 0,C 180,E1 -10735.147,E2 -10735.147} C_VEL
LIN {X 0,Y 405.993,Z 581.81,A -85,B 0,C 180,E1 -10736.47,E2 -10736.47} C_VEL
LIN {X 0,Y 406.878,Z 571.828,A -85,B 0,C 180,E1 -10737.658,E2 -10737.658} C_VEL
LIN {X 0,Y 407.857,Z 560.892,A -85,B 0,C 180,E1 -10738.702,E2 -10738.702} C_VEL
LIN {X 0,Y 408.65,Z 549.504,A -85,B 0,C 180,E1 -10739.561,E2 -10739.561} C_VEL
LIN {X 0,Y 409.444,Z 536.754,A -85,B 0,C 180,E1 -10740.278,E2 -10740.278} C_VEL
LIN {X 0,Y 410.007,Z 523.54,A -85,B 0,C 180,E1 -10740.802,E2 -10740.802} C_VEL
LIN {X 0,Y 410.407,Z 510.062,A -85,B 0,C 180,E1 -10741.115,E2 -10741.115} C_VEL
LIN {X 0,Y 411.451,Z 434.055,A -85,B 0,C 180,E1 -10742.471,E2 -10742.471} C_VEL
LIN {X 0,Y 407.217,Z 413.766,A -85,B 0,C 180,E1 -10743.103,E2 -10743.103} C_VEL
LIN {X 0,Y 406.636,Z 410.823,A -85,B 0,C 180,E1 -10743.25,E2 -10743.25} C_VEL
LIN {X 0,Y 407.077,Z 403.327,A -85,B 0,C 180,E1 -10745.022,E2 -10745.022} C_VEL
LIN {X 0,Y 404.869,Z 391.907,A -85,B 0,C 180,E1 -10748.04,E2 -10748.04} C_VEL
LIN {X 0,Y 404.199,Z 388.676,A -85,B 0,C 180,E1 -10748.991,E2 -10748.991} C_VEL
LIN {X 0,Y 404.207,Z 388.634,A -85,B 0,C 180,E1 -10752.694,E2 -10752.694} C_VEL
LIN {X 0,Y 404.2,Z 388.635,A -85,B 0,C 180,E1 -10755.933,E2 -10755.933} C_VEL
LIN {X 0,Y 404.159,Z 388.636,A -85,B 0,C 180,E1 -10758.64,E2 -10758.64} C_VEL
LIN {X 0,Y 404.157,Z 388.635,A -85,B 0,C 180,E1 -10761.49,E2 -10761.49} C_VEL
LIN {X 0,Y 404.179,Z 388.63,A -85,B 0,C 180,E1 -10764.983,E2 -10764.983} C_VEL
LIN {X 0,Y 404.144,Z 388.643,A -85,B 0,C 180,E1 -10768.554,E2 -10768.554} C_VEL
LIN {X 0,Y 404.191,Z 388.633,A -85,B 0,C 180,E1 -10772,E2 -10772} C_VEL
LIN {X 0,Y 404.17,Z 388.641,A -85,B 0,C 180,E1 -10775.334,E2 -10775.334} C_VEL
LIN {X 0,Y 404.181,Z 388.634,A -85,B 0,C 180,E1 -10778.583,E2 -10778.583} C_VEL
LIN {X 0,Y 404.205,Z 388.629,A -85,B 0,C 180,E1 -10781.762,E2 -10781.762} C_VEL
LIN {X 0,Y 404.199,Z 388.634,A -85,B 0,C 180,E1 -10784.882,E2 -10784.882} C_VEL
LIN {X 0,Y 404.262,Z 388.626,A -85,B 0,C 180,E1 -10787.959,E2 -10787.959} C_VEL
LIN {X 0,Y 404.424,Z 388.606,A -85,B 0,C 180,E1 -10792.1,E2 -10792.1} C_VEL
LIN {X 0,Y 404.416,Z 388.601,A -85,B 0,C 180,E1 -10794.015,E2 -10794.015} C_VEL
LIN {X 0,Y 404.476,Z 388.597,A -85,B 0,C 180,E1 -10798.009,E2 -10798.009} C_VEL
LIN {X 0,Y 404.604,Z 388.579,A -85,B 0,C 180,E1 -10800,E2 -10800} C_VEL
LIN {X 0,Y 404.416,Z 388.604,A -85,B 0,C 180,E1 -10802.989,E2 -10802.989} C_VEL
LIN {X 0,Y 404.403,Z 388.61,A -85,B 0,C 180,E1 -10806.987,E2 -10806.987} C_VEL
LIN {X 0,Y 404.263,Z 388.623,A -85,B 0,C 180,E1 -10810.012,E2 -10810.012} C_VEL
LIN {X 0,Y 404.258,Z 388.62,A -85,B 0,C 180,E1 -10813.212,E2 -10813.212} C_VEL
LIN {X 0,Y 404.207,Z 388.632,A -85,B 0,C 180,E1 -10817.007,E2 -10817.007} C_VEL
LIN {X 0,Y 404.18,Z 388.638,A -85,B 0,C 180,E1 -10820.351,E2 -10820.351} C_VEL
LIN {X 0,Y 404.162,Z 388.636,A -85,B 0,C 180,E1 -10823.575,E2 -10823.575} C_VEL
LIN {X 0,Y 404.176,Z 388.635,A -85,B 0,C 180,E1 -10825.767,E2 -10825.767} C_VEL
LIN {X 0,Y 404.189,Z 388.633,A -85,B 0,C 180,E1 -10828,E2 -10828} C_VEL
LIN {X 0,Y 404.133,Z 388.641,A -85,B 0,C 180,E1 -10831.559,E2 -10831.559} C_VEL
LIN {X 0,Y 404.18,Z 388.639,A -85,B 0,C 180,E1 -10835.017,E2 -10835.017} C_VEL
LIN {X 0,Y 404.158,Z 388.643,A -85,B 0,C 180,E1 -10838.757,E2 -10838.757} C_VEL
LIN {X 0,Y 404.187,Z 388.62,A -85,B 0,C 180,E1 -10841.612,E2 -10841.612} C_VEL
LIN {X 0,Y 404.186,Z 388.639,A -85,B 0,C 180,E1 -10844.529,E2 -10844.529} C_VEL
LIN {X 0,Y 404.136,Z 388.641,A -85,B 0,C 180,E1 -10847.297,E2 -10847.297} C_VEL
LIN {X 0,Y 404.166,Z 388.634,A -85,B 0,C 180,E1 -10849.956,E2 -10849.956} C_VEL
LIN {X 0,Y 404.137,Z 388.637,A -85,B 0,C 180,E1 -10853.125,E2 -10853.125} C_VEL
LIN {X 0,Y 404.143,Z 388.64,A -85,B 0,C 180,E1 -10856.189,E2 -10856.189} C_VEL
LIN {X 0,Y 404.145,Z 388.644,A -85,B 0,C 180,E1 -10859.716,E2 -10859.716} C_VEL
LIN {X 0,Y 404.253,Z 388.777,A -85,B 0,C 180,E1 -10862.141,E2 -10862.141} C_VEL
LIN {X 0,Y 406.569,Z 399.665,A -85,B 0,C 180,E1 -10864.944,E2 -10864.944} C_VEL
LIN {X 0,Y 407.517,Z 405.108,A -85,B 0,C 180,E1 -10866.272,E2 -10866.272} C_VEL
LIN {X 0,Y 407.207,Z 411.374,A -85,B 0,C 180,E1 -10867.686,E2 -10867.686} C_VEL
LIN {X 0,Y 406.449,Z 421.106,A -85,B 0,C 180,E1 -10869.789,E2 -10869.789} C_VEL
LIN {X 0,Y 407.334,Z 425.494,A -85,B 0,C 180,E1 -10869.976,E2 -10869.976} C_VEL
LIN {X 0,Y 410.875,Z 444.814,A -85,B 0,C 180,E1 -10870.547,E2 -10870.547} C_VEL
LIN {X 0,Y 411.251,Z 449.957,A -85,B 0,C 180,E1 -10870.664,E2 -10870.664} C_VEL
LIN {X 0,Y 410.113,Z 529.15,A -85,B 0,C 180,E1 -10872.099,E2 -10872.099} C_VEL
LIN {X 0,Y 409.543,Z 543.001,A -85,B 0,C 180,E1 -10872.557,E2 -10872.557} C_VEL
LIN {X 0,Y 408.858,Z 554.865,A -85,B 0,C 180,E1 -10873.138,E2 -10873.138} C_VEL
LIN {X 0,Y 408.082,Z 566.108,A -85,B 0,C 180,E1 -10873.877,E2 -10873.877} C_VEL
LIN {X 0,Y 407.107,Z 577.722,A -85,B 0,C 180,E1 -10874.865,E2 -10874.865} C_VEL
LIN {X 0,Y 406.215,Z 588.171,A -85,B 0,C 180,E1 -10875.983,E2 -10875.983} C_VEL
LIN {X 0,Y 405.468,Z 597.603,A -85,B 0,C 180,E1 -10877.233,E2 -10877.233} C_VEL
LIN {X 0,Y 404.612,Z 605.349,A -85,B 0,C 180,E1 -10878.478,E2 -10878.478} C_VEL
LIN {X 0,Y 403.987,Z 612.926,A -85,B 0,C 180,E1 -10879.982,E2 -10879.982} C_VEL
LIN {X 0,Y 403.484,Z 619.036,A -85,B 0,C 180,E1 -10881.486,E2 -10881.486} C_VEL
LIN {X 0,Y 403.139,Z 623.894,A -85,B 0,C 180,E1 -10882.991,E2 -10882.991} C_VEL
LIN {X 0,Y 402.98,Z 627.642,A -85,B 0,C 180,E1 -10884.496,E2 -10884.496} C_VEL
LIN {X 0,Y 402.846,Z 630.382,A -85,B 0,C 180,E1 -10885.999,E2 -10885.999} C_VEL
LIN {X 0,Y 402.823,Z 632.588,A -85,B 0,C 180,E1 -10888.001,E2 -10888.001} C_VEL
LIN {X 0,Y 402.845,Z 633.087,A -85,B 0,C 180,E1 -10889.001,E2 -10889.001} C_VEL
LIN {X 0,Y 402.845,Z 632.861,A -85,B 0,C 180,E1 -10891,E2 -10891} C_VEL
LIN {X 0,Y 402.823,Z 632.17,A -85,B 0,C 180,E1 -10892,E2 -10892} C_VEL
LIN {X 0,Y 402.786,Z 631.071,A -85,B 0,C 180,E1 -10893.001,E2 -10893.001} C_VEL
LIN {X 0,Y 402.843,Z 629.524,A -85,B 0,C 180,E1 -10894.002,E2 -10894.002} C_VEL
LIN {X 0,Y 402.938,Z 626.41,A -85,B 0,C 180,E1 -10895.505,E2 -10895.505} C_VEL
LIN {X 0,Y 403.101,Z 622.226,A -85,B 0,C 180,E1 -10897.01,E2 -10897.01} C_VEL
LIN {X 0,Y 403.47,Z 615.841,A -85,B 0,C 180,E1 -10898.767,E2 -10898.767} C_VEL
LIN {X 0,Y 403.933,Z 608.871,A -85,B 0,C 180,E1 -10900.273,E2 -10900.273} C_VEL
LIN {X 0,Y 404.583,Z 600.117,A -85,B 0,C 180,E1 -10901.777,E2 -10901.777} C_VEL
LIN {X 0,Y 405.202,Z 591.133,A -85,B 0,C 180,E1 -10903.031,E2 -10903.031} C_VEL
LIN {X 0,Y 405.961,Z 580.892,A -85,B 0,C 180,E1 -10904.193,E2 -10904.193} C_VEL
LIN {X 0,Y 406.646,Z 570.335,A -85,B 0,C 180,E1 -10905.153,E2 -10905.153} C_VEL
LIN {X 0,Y 407.418,Z 558.068,A -85,B 0,C 180,E1 -10906.022,E2 -10906.022} C_VEL
LIN {X 0,Y 408.074,Z 545.183,A -85,B 0,C 180,E1 -10906.702,E2 -10906.702} C_VEL
LIN {X 0,Y 408.596,Z 532.198,A -85,B 0,C 180,E1 -10907.163,E2 -10907.163} C_VEL
LIN {X 0,Y 408.877,Z 513.785,A -85,B 0,C 180,E1 -10907.538,E2 -10907.538} C_VEL
LIN {X 0,Y 409.621,Z 446.719,A -85,B 0,C 180,E1 -10908.714,E2 -10908.714} C_VEL
LIN {X 0,Y 405.687,Z 421.631,A -85,B 0,C 180,E1 -10909.349,E2 -10909.349} C_VEL
LIN {X 0,Y 405.767,Z 419.381,A -85,B 0,C 180,E1 -10909.739,E2 -10909.739} C_VEL
LIN {X 0,Y 406.838,Z 403.548,A -85,B 0,C 180,E1 -10913.141,E2 -10913.141} C_VEL
LIN {X 0,Y 405.432,Z 394.947,A -85,B 0,C 180,E1 -10915.116,E2 -10915.116} C_VEL
LIN {X 0,Y 404.278,Z 388.793,A -85,B 0,C 180,E1 -10916.592,E2 -10916.592} C_VEL
LIN {X 0,Y 404.146,Z 388.641,A -85,B 0,C 180,E1 -10920.285,E2 -10920.285} C_VEL
LIN {X 0,Y 404.145,Z 388.643,A -85,B 0,C 180,E1 -10923.812,E2 -10923.812} C_VEL
LIN {X 0,Y 404.14,Z 388.641,A -85,B 0,C 180,E1 -10926.875,E2 -10926.875} C_VEL
LIN {X 0,Y 404.148,Z 388.641,A -85,B 0,C 180,E1 -10930.08,E2 -10930.08} C_VEL
LIN {X 0,Y 404.155,Z 388.641,A -85,B 0,C 180,E1 -10933.084,E2 -10933.084} C_VEL
LIN {X 0,Y 404.2,Z 388.635,A -85,B 0,C 180,E1 -10935.933,E2 -10935.933} C_VEL
LIN {X 0,Y 404.162,Z 388.638,A -85,B 0,C 180,E1 -10938.64,E2 -10938.64} C_VEL
LIN {X 0,Y 404.16,Z 388.643,A -85,B 0,C 180,E1 -10941.49,E2 -10941.49} C_VEL
LIN {X 0,Y 404.182,Z 388.638,A -85,B 0,C 180,E1 -10944.983,E2 -10944.983} C_VEL
LIN {X 0,Y 404.138,Z 388.641,A -85,B 0,C 180,E1 -10948.553,E2 -10948.553} C_VEL
LIN {X 0,Y 404.191,Z 388.636,A -85,B 0,C 180,E1 -10952,E2 -10952} C_VEL
LIN {X 0,Y 404.17,Z 388.642,A -85,B 0,C 180,E1 -10955.334,E2 -10955.334} C_VEL
LIN {X 0,Y 404.133,Z 388.642,A -85,B 0,C 180,E1 -10958.58,E2 -10958.58} C_VEL
LIN {X 0,Y 404.205,Z 388.636,A -85,B 0,C 180,E1 -10961.762,E2 -10961.762} C_VEL
LIN {X 0,Y 404.2,Z 388.636,A -85,B 0,C 180,E1 -10964.882,E2 -10964.882} C_VEL
LIN {X 0,Y 404.251,Z 388.629,A -85,B 0,C 180,E1 -10967.958,E2 -10967.958} C_VEL
LIN {X 0,Y 404.4,Z 388.609,A -85,B 0,C 180,E1 -10972.129,E2 -10972.129} C_VEL
LIN {X 0,Y 404.417,Z 388.608,A -85,B 0,C 180,E1 -10974.015,E2 -10974.015} C_VEL
LIN {X 0,Y 404.477,Z 388.6,A -85,B 0,C 180,E1 -10978.008,E2 -10978.008} C_VEL
LIN {X 0,Y 404.605,Z 388.584,A -85,B 0,C 180,E1 -10980,E2 -10980} C_VEL
LIN {X 0,Y 404.418,Z 388.611,A -85,B 0,C 180,E1 -10982.988,E2 -10982.988} C_VEL
LIN {X 0,Y 404.401,Z 388.613,A -85,B 0,C 180,E1 -10986.987,E2 -10986.987} C_VEL
LIN {X 0,Y 404.253,Z 388.628,A -85,B 0,C 180,E1 -10990.012,E2 -10990.012} C_VEL
LIN {X 0,Y 404.261,Z 388.63,A -85,B 0,C 180,E1 -10993.211,E2 -10993.211} C_VEL
LIN {X 0,Y 404.21,Z 388.636,A -85,B 0,C 180,E1 -10997.007,E2 -10997.007} C_VEL
LIN {X 0,Y 404.159,Z 388.639,A -85,B 0,C 180,E1 -11000.352,E2 -11000.352} C_VEL
LIN {X 0,Y 404.164,Z 388.641,A -85,B 0,C 180,E1 -11003.575,E2 -11003.575} C_VEL
LIN {X 0,Y 404.179,Z 388.638,A -85,B 0,C 180,E1 -11005.767,E2 -11005.767} C_VEL
LIN {X 0,Y 404.194,Z 388.635,A -85,B 0,C 180,E1 -11008,E2 -11008} C_VEL
LIN {X 0,Y 404.14,Z 388.644,A -85,B 0,C 180,E1 -11011.56,E2 -11011.56} C_VEL
LIN {X 0,Y 404.182,Z 388.639,A -85,B 0,C 180,E1 -11015.016,E2 -11015.016} C_VEL
LIN {X 0,Y 404.154,Z 388.642,A -85,B 0,C 180,E1 -11018.757,E2 -11018.757} C_VEL
LIN {X 0,Y 404.121,Z 388.645,A -85,B 0,C 180,E1 -11021.6,E2 -11021.6} C_VEL
LIN {X 0,Y 404.146,Z 388.642,A -85,B 0,C 180,E1 -11024.523,E2 -11024.523} C_VEL
LIN {X 0,Y 404.169,Z 388.642,A -85,B 0,C 180,E1 -11027.301,E2 -11027.301} C_VEL
LIN {X 0,Y 404.167,Z 388.638,A -85,B 0,C 180,E1 -11029.956,E2 -11029.956} C_VEL
LIN {X 0,Y 404.14,Z 388.647,A -85,B 0,C 180,E1 -11033.125,E2 -11033.125} C_VEL
LIN {X 0,Y 404.144,Z 388.64,A -85,B 0,C 180,E1 -11036.188,E2 -11036.188} C_VEL
LIN {X 0,Y 404.145,Z 388.64,A -85,B 0,C 180,E1 -11039.715,E2 -11039.715} C_VEL
LIN {X 0,Y 404.196,Z 388.639,A -85,B 0,C 180,E1 -11043.123,E2 -11043.123} C_VEL
LIN {X 0,Y 404.178,Z 388.639,A -85,B 0,C 180,E1 -11045.335,E2 -11045.335} C_VEL
LIN {X 0,Y 404.139,Z 388.643,A -85,B 0,C 180,E1 -11048.581,E2 -11048.581} C_VEL
LIN {X 0,Y 404.211,Z 388.631,A -85,B 0,C 180,E1 -11051.762,E2 -11051.762} C_VEL
LIN {X 0,Y 404.208,Z 388.638,A -85,B 0,C 180,E1 -11054.882,E2 -11054.882} C_VEL
LIN {X 0,Y 404.258,Z 388.63,A -85,B 0,C 180,E1 -11057.959,E2 -11057.959} C_VEL
LIN {X 0,Y 404.31,Z 388.855,A -85,B 0,C 180,E1 -11058.437,E2 -11058.437} C_VEL
LIN {X 0,Y 406.321,Z 400.307,A -85,B 0,C 180,E1 -11061.295,E2 -11061.295} C_VEL
LIN {X 0,Y 405.83,Z 406.741,A -85,B 0,C 180,E1 -11062.787,E2 -11062.787} C_VEL
LIN {X 0,Y 405.66,Z 410.901,A -85,B 0,C 180,E1 -11063.69,E2 -11063.69} C_VEL
LIN {X 0,Y 406.425,Z 415.559,A -85,B 0,C 180,E1 -11063.847,E2 -11063.847} C_VEL
LIN {X 0,Y 409.773,Z 433.657,A -85,B 0,C 180,E1 -11064.308,E2 -11064.308} C_VEL
LIN {X 0,Y 408.721,Z 517.793,A -85,B 0,C 180,E1 -11065.801,E2 -11065.801} C_VEL
LIN {X 0,Y 408.301,Z 530.461,A -85,B 0,C 180,E1 -11066.206,E2 -11066.206} C_VEL
LIN {X 0,Y 407.716,Z 543.848,A -85,B 0,C 180,E1 -11066.85,E2 -11066.85} C_VEL
LIN {X 0,Y 407.022,Z 555.899,A -85,B 0,C 180,E1 -11067.65,E2 -11067.65} C_VEL
LIN {X 0,Y 406.237,Z 567.374,A -85,B 0,C 180,E1 -11068.637,E2 -11068.637} C_VEL
LIN {X 0,Y 405.477,Z 577.714,A -85,B 0,C 180,E1 -11069.751,E2 -11069.751} C_VEL
LIN {X 0,Y 405.034,Z 583.369,A -85,B 0,C 180,E1 -11070.478,E2 -11070.478} C_VEL
LIN {X 0,Y 404.117,Z 587.55,A -85,B 0,C 180,E1 -11071.055,E2 -11071.055} C_VEL
LIN {X 0,Y 400.802,Z 593.941,A -85,B 0,C 180,E1 -11072.029,E2 -11072.029} C_VEL
LIN {X 0,Y 397.496,Z 599.756,A -85,B 0,C 180,E1 -11073.086,E2 -11073.086} C_VEL
LIN {X 0,Y 396.603,Z 602.981,A -85,B 0,C 180,E1 -11073.786,E2 -11073.786} C_VEL
LIN {X 0,Y 396.229,Z 608.067,A -85,B 0,C 180,E1 -11075.088,E2 -11075.088} C_VEL
LIN {X 0,Y 396.075,Z 612.41,A -85,B 0,C 180,E1 -11076.45,E2 -11076.45} C_VEL
LIN {X 0,Y 395.85,Z 616.616,A -85,B 0,C 180,E1 -11078.165,E2 -11078.165} C_VEL
LIN {X 0,Y 395.72,Z 618.543,A -85,B 0,C 180,E1 -11079.197,E2 -11079.197} C_VEL
LIN {X 0,Y 395.644,Z 620.011,A -85,B 0,C 180,E1 -11080.232,E2 -11080.232} C_VEL
LIN {X 0,Y 395.65,Z 621.043,A -85,B 0,C 180,E1 -11081.267,E2 -11081.267} C_VEL
LIN {X 0,Y 395.688,Z 621.698,A -85,B 0,C 180,E1 -11082.344,E2 -11082.344} C_VEL
LIN {X 0,Y 395.578,Z 621.922,A -85,B 0,C 180,E1 -11083.353,E2 -11083.353} C_VEL
LIN {X 0,Y 395.567,Z 621.707,A -85,B 0,C 180,E1 -11084.402,E2 -11084.402} C_VEL
LIN {X 0,Y 395.688,Z 620.122,A -85,B 0,C 180,E1 -11086.439,E2 -11086.439} C_VEL
LIN {X 0,Y 395.804,Z 618.558,A -85,B 0,C 180,E1 -11087.568,E2 -11087.568} C_VEL
LIN {X 0,Y 396.049,Z 615.445,A -85,B 0,C 180,E1 -11089.164,E2 -11089.164} C_VEL
LIN {X 0,Y 396.354,Z 611.176,A -85,B 0,C 180,E1 -11090.77,E2 -11090.77} C_VEL
LIN {X 0,Y 396.928,Z 604.562,A -85,B 0,C 180,E1 -11092.65,E2 -11092.65} C_VEL
LIN {X 0,Y 397.649,Z 597.245,A -85,B 0,C 180,E1 -11094.262,E2 -11094.262} C_VEL
LIN {X 0,Y 398.56,Z 588.264,A -85,B 0,C 180,E1 -11095.828,E2 -11095.828} C_VEL
LIN {X 0,Y 399.49,Z 578.357,A -85,B 0,C 180,E1 -11097.219,E2 -11097.219} C_VEL
LIN {X 0,Y 400.538,Z 567.55,A -85,B 0,C 180,E1 -11098.416,E2 -11098.416} C_VEL
LIN {X 0,Y 401.372,Z 556.979,A -85,B 0,C 180,E1 -11099.358,E2 -11099.358} C_VEL
LIN {X 0,Y 402.25,Z 545.593,A -85,B 0,C 180,E1 -11100.152,E2 -11100.152} C_VEL
LIN {X 0,Y 402.963,Z 532.777,A -85,B 0,C 180,E1 -11100.816,E2 -11100.816} C_VEL
LIN {X 0,Y 403.534,Z 519.404,A -85,B 0,C 180,E1 -11101.278,E2 -11101.278} C_VEL
LIN {X 0,Y 404.165,Z 480.071,A -85,B 0,C 180,E1 -11102.024,E2 -11102.024} C_VEL
LIN {X 0,Y 404.856,Z 434.678,A -85,B 0,C 180,E1 -11102.846,E2 -11102.846} C_VEL
LIN {X 0,Y 400.428,Z 413.926,A -85,B 0,C 180,E1 -11103.515,E2 -11103.515} C_VEL
LIN {X 0,Y 399.812,Z 411.021,A -85,B 0,C 180,E1 -11103.659,E2 -11103.659} C_VEL
LIN {X 0,Y 400.188,Z 404.926,A -85,B 0,C 180,E1 -11105.112,E2 -11105.112} C_VEL
LIN {X 0,Y 398.006,Z 393.55,A -85,B 0,C 180,E1 -11108.171,E2 -11108.171} C_VEL
LIN {X 0,Y 397.167,Z 389.56,A -85,B 0,C 180,E1 -11109.35,E2 -11109.35} C_VEL
LIN {X 0,Y 397.156,Z 389.515,A -85,B 0,C 180,E1 -11112.254,E2 -11112.254} C_VEL
LIN {X 0,Y 397.145,Z 389.512,A -85,B 0,C 180,E1 -11115.059,E2 -11115.059} C_VEL
LIN {X 0,Y 397.15,Z 389.506,A -85,B 0,C 180,E1 -11118.006,E2 -11118.006} C_VEL
LIN {X 0,Y 397.104,Z 389.514,A -85,B 0,C 180,E1 -11121.725,E2 -11121.725} C_VEL
LIN {X 0,Y 397.119,Z 389.508,A -85,B 0,C 180,E1 -11125.506,E2 -11125.506} C_VEL
LIN {X 0,Y 397.081,Z 389.514,A -85,B 0,C 180,E1 -11129.118,E2 -11129.118} C_VEL
LIN {X 0,Y 397.187,Z 389.509,A -85,B 0,C 180,E1 -11132.609,E2 -11132.609} C_VEL
LIN {X 0,Y 397.126,Z 389.515,A -85,B 0,C 180,E1 -11135.981,E2 -11135.981} C_VEL
LIN {X 0,Y 397.159,Z 389.511,A -85,B 0,C 180,E1 -11139.693,E2 -11139.693} C_VEL
LIN {X 0,Y 397.173,Z 389.51,A -85,B 0,C 180,E1 -11142.845,E2 -11142.845} C_VEL
LIN {X 0,Y 397.218,Z 389.503,A -85,B 0,C 180,E1 -11146.679,E2 -11146.679} C_VEL
LIN {X 0,Y 397.221,Z 389.495,A -85,B 0,C 180,E1 -11149.809,E2 -11149.809} C_VEL
LIN {X 0,Y 397.356,Z 389.488,A -85,B 0,C 180,E1 -11152.888,E2 -11152.888} C_VEL
LIN {X 0,Y 397.25,Z 389.497,A -85,B 0,C 180,E1 -11154.925,E2 -11154.925} C_VEL
LIN {X 0,Y 397.445,Z 389.473,A -85,B 0,C 180,E1 -11157.973,E2 -11157.973} C_VEL
LIN {X 0,Y 397.574,Z 389.455,A -85,B 0,C 180,E1 -11160,E2 -11160} C_VEL
LIN {X 0,Y 397.375,Z 389.48,A -85,B 0,C 180,E1 -11163.042,E2 -11163.042} C_VEL
LIN {X 0,Y 397.356,Z 389.486,A -85,B 0,C 180,E1 -11167.112,E2 -11167.112} C_VEL
LIN {X 0,Y 397.221,Z 389.501,A -85,B 0,C 180,E1 -11170.191,E2 -11170.191} C_VEL
LIN {X 0,Y 397.218,Z 389.496,A -85,B 0,C 180,E1 -11173.321,E2 -11173.321} C_VEL
LIN {X 0,Y 397.174,Z 389.506,A -85,B 0,C 180,E1 -11177.156,E2 -11177.156} C_VEL
LIN {X 0,Y 397.107,Z 389.521,A -85,B 0,C 180,E1 -11180.73,E2 -11180.73} C_VEL
LIN {X 0,Y 397.126,Z 389.513,A -85,B 0,C 180,E1 -11184.019,E2 -11184.019} C_VEL
LIN {X 0,Y 397.187,Z 389.505,A -85,B 0,C 180,E1 -11187.391,E2 -11187.391} C_VEL
LIN {X 0,Y 397.072,Z 389.521,A -85,B 0,C 180,E1 -11190.883,E2 -11190.883} C_VEL
LIN {X 0,Y 397.12,Z 389.516,A -85,B 0,C 180,E1 -11194.494,E2 -11194.494} C_VEL
LIN {X 0,Y 397.105,Z 389.518,A -85,B 0,C 180,E1 -11198.275,E2 -11198.275} C_VEL
LIN {X 0,Y 397.151,Z 389.498,A -85,B 0,C 180,E1 -11201.994,E2 -11201.994} C_VEL
LIN {X 0,Y 397.109,Z 389.514,A -85,B 0,C 180,E1 -11205.066,E2 -11205.066} C_VEL
LIN {X 0,Y 397.076,Z 389.522,A -85,B 0,C 180,E1 -11208.02,E2 -11208.02} C_VEL
LIN {X 0,Y 397.13,Z 389.517,A -85,B 0,C 180,E1 -11211.139,E2 -11211.139} C_VEL
LIN {X 0,Y 397.118,Z 389.518,A -85,B 0,C 180,E1 -11214.497,E2 -11214.497} C_VEL
LIN {X 0,Y 397.077,Z 389.523,A -85,B 0,C 180,E1 -11217.929,E2 -11217.929} C_VEL
LIN {X 0,Y 397.179,Z 389.588,A -85,B 0,C 180,E1 -11221.721,E2 -11221.721} C_VEL
LIN {X 0,Y 399.157,Z 398.556,A -85,B 0,C 180,E1 -11224.129,E2 -11224.129} C_VEL
LIN {X 0,Y 400.652,Z 406.868,A -85,B 0,C 180,E1 -11226.207,E2 -11226.207} C_VEL
LIN {X 0,Y 400.085,Z 415.1,A -85,B 0,C 180,E1 -11228.083,E2 -11228.083} C_VEL
LIN {X 0,Y 399.626,Z 421.181,A -85,B 0,C 180,E1 -11229.386,E2 -11229.386} C_VEL
LIN {X 0,Y 401.488,Z 430.239,A -85,B 0,C 180,E1 -11229.714,E2 -11229.714} C_VEL
LIN {X 0,Y 404.618,Z 447.579,A -85,B 0,C 180,E1 -11230.235,E2 -11230.235} C_VEL
LIN {X 0,Y 403.71,Z 519.061,A -85,B 0,C 180,E1 -11231.537,E2 -11231.537} C_VEL
LIN {X 0,Y 403.371,Z 533.156,A -85,B 0,C 180,E1 -11231.855,E2 -11231.855} C_VEL
LIN {X 0,Y 402.718,Z 546.172,A -85,B 0,C 180,E1 -11232.35,E2 -11232.35} C_VEL
LIN {X 0,Y 402.016,Z 557.619,A -85,B 0,C 180,E1 -11232.974,E2 -11232.974} C_VEL
LIN {X 0,Y 401.014,Z 569.78,A -85,B 0,C 180,E1 -11233.847,E2 -11233.847} C_VEL
LIN {X 0,Y 400.065,Z 580.562,A -85,B 0,C 180,E1 -11234.842,E2 -11234.842} C_VEL
LIN {X 0,Y 399.173,Z 590.485,A -85,B 0,C 180,E1 -11235.991,E2 -11235.991} C_VEL
LIN {X 0,Y 398.367,Z 599.434,A -85,B 0,C 180,E1 -11237.261,E2 -11237.261} C_VEL
LIN {X 0,Y 397.413,Z 608.199,A -85,B 0,C 180,E1 -11238.783,E2 -11238.783} C_VEL
LIN {X 0,Y 396.785,Z 615.226,A -85,B 0,C 180,E1 -11240.313,E2 -11240.313} C_VEL
LIN {X 0,Y 396.305,Z 620.852,A -85,B 0,C 180,E1 -11241.844,E2 -11241.844} C_VEL
LIN {X 0,Y 395.954,Z 626.101,A -85,B 0,C 180,E1 -11243.709,E2 -11243.709} C_VEL
LIN {X 0,Y 395.887,Z 628.666,A -85,B 0,C 180,E1 -11244.908,E2 -11244.908} C_VEL
LIN {X 0,Y 395.692,Z 631.631,A -85,B 0,C 180,E1 -11246.946,E2 -11246.946} C_VEL
LIN {X 0,Y 395.719,Z 632.524,A -85,B 0,C 180,E1 -11247.965,E2 -11247.965} C_VEL
LIN {X 0,Y 395.756,Z 632.994,A -85,B 0,C 180,E1 -11248.983,E2 -11248.983} C_VEL
LIN {X 0,Y 395.76,Z 633.058,A -85,B 0,C 180,E1 -11250,E2 -11250} C_VEL
LIN {X 0,Y 395.756,Z 632.738,A -85,B 0,C 180,E1 -11251.018,E2 -11251.018} C_VEL
LIN {X 0,Y 395.72,Z 632.033,A -85,B 0,C 180,E1 -11252.036,E2 -11252.036} C_VEL
LIN {X 0,Y 395.692,Z 630.903,A -85,B 0,C 180,E1 -11253.055,E2 -11253.055} C_VEL
LIN {X 0,Y 395.767,Z 629.34,A -85,B 0,C 180,E1 -11254.073,E2 -11254.073} C_VEL
LIN {X 0,Y 395.842,Z 625.648,A -85,B 0,C 180,E1 -11255.826,E2 -11255.826} C_VEL
LIN {X 0,Y 396.139,Z 620.338,A -85,B 0,C 180,E1 -11257.647,E2 -11257.647} C_VEL
LIN {X 0,Y 396.551,Z 613.36,A -85,B 0,C 180,E1 -11259.435,E2 -11259.435} C_VEL
LIN {X 0,Y 397.066,Z 605.796,A -85,B 0,C 180,E1 -11260.969,E2 -11260.969} C_VEL
LIN {X 0,Y 397.72,Z 598.069,A -85,B 0,C 180,E1 -11262.242,E2 -11262.242} C_VEL
LIN {X 0,Y 398.425,Z 588.819,A -85,B 0,C 180,E1 -11263.494,E2 -11263.494} C_VEL
LIN {X 0,Y 399.186,Z 578.267,A -85,B 0,C 180,E1 -11264.647,E2 -11264.647} C_VEL
LIN {X 0,Y 399.946,Z 566.449,A -85,B 0,C 180,E1 -11265.675,E2 -11265.675} C_VEL
LIN {X 0,Y 400.771,Z 554.026,A -85,B 0,C 180,E1 -11266.491,E2 -11266.491} C_VEL
LIN {X 0,Y 401.363,Z 540.906,A -85,B 0,C 180,E1 -11267.121,E2 -11267.121} C_VEL
LIN {X 0,Y 401.819,Z 527.987,A -85,B 0,C 180,E1 -11267.527,E2 -11267.527} C_VEL
LIN {X 0,Y 402.697,Z 446.905,A -85,B 0,C 180,E1 -11268.992,E2 -11268.992} C_VEL
LIN {X 0,Y 398.74,Z 421.435,A -85,B 0,C 180,E1 -11269.649,E2 -11269.649} C_VEL
LIN {X 0,Y 398.921,Z 417.806,A -85,B 0,C 180,E1 -11270.362,E2 -11270.362} C_VEL
LIN {X 0,Y 399.873,Z 404.405,A -85,B 0,C 180,E1 -11273.294,E2 -11273.294} C_VEL
LIN {X 0,Y 398.053,Z 393.824,A -85,B 0,C 180,E1 -11275.782,E2 -11275.782} C_VEL
LIN {X 0,Y 397.202,Z 389.599,A -85,B 0,C 180,E1 -11276.855,E2 -11276.855} C_VEL
LIN {X 0,Y 397.106,Z 389.52,A -85,B 0,C 180,E1 -11279.864,E2 -11279.864} C_VEL
LIN {X 0,Y 397.119,Z 389.519,A -85,B 0,C 180,E1 -11283.717,E2 -11283.717} C_VEL
LIN {X 0,Y 397.097,Z 389.521,A -85,B 0,C 180,E1 -11287.209,E2 -11287.209} C_VEL
LIN {X 0,Y 397.102,Z 389.517,A -85,B 0,C 180,E1 -11290.445,E2 -11290.445} C_VEL
LIN {X 0,Y 397.104,Z 389.521,A -85,B 0,C 180,E1 -11293.647,E2 -11293.647} C_VEL
LIN {X 0,Y 397.158,Z 389.51,A -85,B 0,C 180,E1 -11296.512,E2 -11296.512} C_VEL
LIN {X 0,Y 397.122,Z 389.519,A -85,B 0,C 180,E1 -11299.55,E2 -11299.55} C_VEL
LIN {X 0,Y 397.096,Z 389.519,A -85,B 0,C 180,E1 -11302.789,E2 -11302.789} C_VEL
LIN {X 0,Y 397.115,Z 389.516,A -85,B 0,C 180,E1 -11306.282,E2 -11306.282} C_VEL
LIN {X 0,Y 397.101,Z 389.518,A -85,B 0,C 180,E1 -11310.135,E2 -11310.135} C_VEL
LIN {X 0,Y 397.19,Z 389.507,A -85,B 0,C 180,E1 -11312.609,E2 -11312.609} C_VEL
LIN {X 0,Y 397.125,Z 389.516,A -85,B 0,C 180,E1 -11315.981,E2 -11315.981} C_VEL
LIN {X 0,Y 397.134,Z 389.517,A -85,B 0,C 180,E1 -11319.704,E2 -11319.704} C_VEL
LIN {X 0,Y 397.177,Z 389.51,A -85,B 0,C 180,E1 -11322.845,E2 -11322.845} C_VEL
LIN {X 0,Y 397.224,Z 389.504,A -85,B 0,C 180,E1 -11326.702,E2 -11326.702} C_VEL
LIN {X 0,Y 397.212,Z 389.506,A -85,B 0,C 180,E1 -11329.809,E2 -11329.809} C_VEL
LIN {X 0,Y 397.347,Z 389.49,A -85,B 0,C 180,E1 -11332.888,E2 -11332.888} C_VEL
LIN {X 0,Y 397.25,Z 389.502,A -85,B 0,C 180,E1 -11334.925,E2 -11334.925} C_VEL
LIN {X 0,Y 397.446,Z 389.476,A -85,B 0,C 180,E1 -11337.973,E2 -11337.973} C_VEL
LIN {X 0,Y 397.575,Z 389.46,A -85,B 0,C 180,E1 -11340,E2 -11340} C_VEL
LIN {X 0,Y 397.377,Z 389.488,A -85,B 0,C 180,E1 -11343.041,E2 -11343.041} C_VEL
LIN {X 0,Y 397.343,Z 389.488,A -85,B 0,C 180,E1 -11346.652,E2 -11346.652} C_VEL
LIN {X 0,Y 397.247,Z 389.504,A -85,B 0,C 180,E1 -11349.162,E2 -11349.162} C_VEL
LIN {X 0,Y 397.214,Z 389.504,A -85,B 0,C 180,E1 -11352.258,E2 -11352.258} C_VEL
LIN {X 0,Y 397.173,Z 389.513,A -85,B 0,C 180,E1 -11355.392,E2 -11355.392} C_VEL
LIN {X 0,Y 397.157,Z 389.512,A -85,B 0,C 180,E1 -11358.574,E2 -11358.574} C_VEL
LIN {X 0,Y 397.092,Z 389.52,A -85,B 0,C 180,E1 -11361.819,E2 -11361.819} C_VEL
LIN {X 0,Y 397.152,Z 389.516,A -85,B 0,C 180,E1 -11365.132,E2 -11365.132} C_VEL
LIN {X 0,Y 397.159,Z 389.512,A -85,B 0,C 180,E1 -11367.777,E2 -11367.777} C_VEL
LIN {X 0,Y 397.082,Z 389.524,A -85,B 0,C 180,E1 -11370.882,E2 -11370.882} C_VEL
LIN {X 0,Y 397.122,Z 389.516,A -85,B 0,C 180,E1 -11374.494,E2 -11374.494} C_VEL
LIN {X 0,Y 397.103,Z 389.518,A -85,B 0,C 180,E1 -11378.275,E2 -11378.275} C_VEL
LIN {X 0,Y 397.086,Z 389.523,A -85,B 0,C 180,E1 -11380.909,E2 -11380.909} C_VEL
LIN {X 0,Y 397.101,Z 389.519,A -85,B 0,C 180,E1 -11383.649,E2 -11383.649} C_VEL
LIN {X 0,Y 397.102,Z 389.519,A -85,B 0,C 180,E1 -11386.521,E2 -11386.521} C_VEL
LIN {X 0,Y 397.119,Z 389.517,A -85,B 0,C 180,E1 -11389.552,E2 -11389.552} C_VEL
LIN {X 0,Y 397.098,Z 389.521,A -85,B 0,C 180,E1 -11392.79,E2 -11392.79} C_VEL
LIN {X 0,Y 397.118,Z 389.516,A -85,B 0,C 180,E1 -11396.282,E2 -11396.282} C_VEL
LIN {X 0,Y 397.105,Z 389.517,A -85,B 0,C 180,E1 -11400.136,E2 -11400.136} C_VEL
LIN {X 0,Y 397.194,Z 389.508,A -85,B 0,C 180,E1 -11402.61,E2 -11402.61} C_VEL
LIN {X 0,Y 397.133,Z 389.513,A -85,B 0,C 180,E1 -11405.982,E2 -11405.982} C_VEL
LIN {X 0,Y 397.139,Z 389.513,A -85,B 0,C 180,E1 -11409.705,E2 -11409.705} C_VEL
LIN {X 0,Y 397.183,Z 389.512,A -85,B 0,C 180,E1 -11412.845,E2 -11412.845} C_VEL
LIN {X 0,Y 397.23,Z 389.505,A -85,B 0,C 180,E1 -11416.703,E2 -11416.703} C_VEL
LIN {X 0,Y 397.233,Z 389.723,A -85,B 0,C 180,E1 -11418.228,E2 -11418.228} C_VEL
LIN {X 0,Y 399.32,Z 401.185,A -85,B 0,C 180,E1 -11421.141,E2 -11421.141} C_VEL
LIN {X 0,Y 398.851,Z 407.629,A -85,B 0,C 180,E1 -11422.66,E2 -11422.66} C_VEL
LIN {X 0,Y 398.801,Z 410.954,A -85,B 0,C 180,E1 -11423.391,E2 -11423.391} C_VEL
LIN {X 0,Y 399.509,Z 416.163,A -85,B 0,C 180,E1 -11423.564,E2 -11423.564} C_VEL
LIN {X 0,Y 402.935,Z 434.243,A -85,B 0,C 180,E1 -11424.037,E2 -11424.037} C_VEL
LIN {X 0,Y 401.843,Z 518.832,A -85,B 0,C 180,E1 -11425.572,E2 -11425.572} C_VEL
LIN {X 0,Y 401.394,Z 531.928,A -85,B 0,C 180,E1 -11426.015,E2 -11426.015} C_VEL
LIN {X 0,Y 400.792,Z 544.924,A -85,B 0,C 180,E1 -11426.67,E2 -11426.67} C_VEL
LIN {X 0,Y 400.052,Z 556.719,A -85,B 0,C 180,E1 -11427.483,E2 -11427.483} C_VEL
LIN {X 0,Y 399.245,Z 568.062,A -85,B 0,C 180,E1 -11428.487,E2 -11428.487} C_VEL
LIN {X 0,Y 398.467,Z 578.294,A -85,B 0,C 180,E1 -11429.621,E2 -11429.621} C_VEL
LIN {X 0,Y 397.822,Z 586.667,A -85,B 0,C 180,E1 -11430.759,E2 -11430.759} C_VEL
LIN {X 0,Y 397.085,Z 595.76,A -85,B 0,C 180,E1 -11432.282,E2 -11432.282} C_VEL
LIN {X 0,Y 396.603,Z 602.981,A -85,B 0,C 180,E1 -11433.786,E2 -11433.786} C_VEL
LIN {X 0,Y 395.759,Z 606.032,A -85,B 0,C 180,E1 -11434.508,E2 -11434.508} C_VEL
LIN {X 0,Y 392.672,Z 610.494,A -85,B 0,C 180,E1 -11435.716,E2 -11435.716} C_VEL
LIN {X 0,Y 389.602,Z 614.203,A -85,B 0,C 180,E1 -11436.993,E2 -11436.993} C_VEL
LIN {X 0,Y 388.801,Z 616.078,A -85,B 0,C 180,E1 -11437.814,E2 -11437.814} C_VEL
LIN {X 0,Y 388.62,Z 618.945,A -85,B 0,C 180,E1 -11439.367,E2 -11439.367} C_VEL
LIN {X 0,Y 388.559,Z 621.293,A -85,B 0,C 180,E1 -11441.476,E2 -11441.476} C_VEL
LIN {X 0,Y 388.574,Z 621.87,A -85,B 0,C 180,E1 -11442.535,E2 -11442.535} C_VEL
LIN {X 0,Y 388.469,Z 622.004,A -85,B 0,C 180,E1 -11443.602,E2 -11443.602} C_VEL
LIN {X 0,Y 388.469,Z 621.719,A -85,B 0,C 180,E1 -11444.671,E2 -11444.671} C_VEL
LIN {X 0,Y 388.596,Z 620.216,A -85,B 0,C 180,E1 -11446.557,E2 -11446.557} C_VEL
LIN {X 0,Y 388.84,Z 617.386,A -85,B 0,C 180,E1 -11448.439,E2 -11448.439} C_VEL
LIN {X 0,Y 389.141,Z 613.699,A -85,B 0,C 180,E1 -11450.093,E2 -11450.093} C_VEL
LIN {X 0,Y 389.555,Z 608.932,A -85,B 0,C 180,E1 -11451.705,E2 -11451.705} C_VEL
LIN {X 0,Y 390.182,Z 602.729,A -85,B 0,C 180,E1 -11453.344,E2 -11453.344} C_VEL
LIN {X 0,Y 390.974,Z 594.916,A -85,B 0,C 180,E1 -11454.987,E2 -11454.987} C_VEL
LIN {X 0,Y 391.861,Z 586.938,A -85,B 0,C 180,E1 -11456.339,E2 -11456.339} C_VEL
LIN {X 0,Y 392.736,Z 577.989,A -85,B 0,C 180,E1 -11457.582,E2 -11457.582} C_VEL
LIN {X 0,Y 393.715,Z 568.394,A -85,B 0,C 180,E1 -11458.667,E2 -11458.667} C_VEL
LIN {X 0,Y 394.762,Z 556.291,A -85,B 0,C 180,E1 -11459.761,E2 -11459.761} C_VEL
LIN {X 0,Y 395.647,Z 544.793,A -85,B 0,C 180,E1 -11460.561,E2 -11460.561} C_VEL
LIN {X 0,Y 396.399,Z 531.919,A -85,B 0,C 180,E1 -11461.218,E2 -11461.218} C_VEL
LIN {X 0,Y 396.959,Z 519.03,A -85,B 0,C 180,E1 -11461.66,E2 -11461.66} C_VEL
LIN {X 0,Y 398.294,Z 435.512,A -85,B 0,C 180,E1 -11463.229,E2 -11463.229} C_VEL
LIN {X 0,Y 393.759,Z 414.549,A -85,B 0,C 180,E1 -11463.927,E2 -11463.927} C_VEL
LIN {X 0,Y 393.042,Z 411.039,A -85,B 0,C 180,E1 -11464.11,E2 -11464.11} C_VEL
LIN {X 0,Y 393.298,Z 406.592,A -85,B 0,C 180,E1 -11465.189,E2 -11465.189} C_VEL
LIN {X 0,Y 391.493,Z 396.923,A -85,B 0,C 180,E1 -11467.826,E2 -11467.826} C_VEL
LIN {X 0,Y 390.093,Z 390.441,A -85,B 0,C 180,E1 -11469.734,E2 -11469.734} C_VEL
LIN {X 0,Y 390.114,Z 390.389,A -85,B 0,C 180,E1 -11473.201,E2 -11473.201} C_VEL
LIN {X 0,Y 390.109,Z 390.394,A -85,B 0,C 180,E1 -11476.797,E2 -11476.797} C_VEL
LIN {X 0,Y 390.073,Z 390.397,A -85,B 0,C 180,E1 -11479.563,E2 -11479.563} C_VEL
LIN {X 0,Y 390.042,Z 390.396,A -85,B 0,C 180,E1 -11482.448,E2 -11482.448} C_VEL
LIN {X 0,Y 390.061,Z 390.389,A -85,B 0,C 180,E1 -11486.045,E2 -11486.045} C_VEL
LIN {X 0,Y 390.042,Z 390.4,A -85,B 0,C 180,E1 -11488.497,E2 -11488.497} C_VEL
LIN {X 0,Y 390.11,Z 390.388,A -85,B 0,C 180,E1 -11492.069,E2 -11492.069} C_VEL
LIN {X 0,Y 390.073,Z 390.396,A -85,B 0,C 180,E1 -11495.519,E2 -11495.519} C_VEL
LIN {X 0,Y 390.083,Z 390.393,A -85,B 0,C 180,E1 -11498.879,E2 -11498.879} C_VEL
LIN {X 0,Y 390.122,Z 390.383,A -85,B 0,C 180,E1 -11502.167,E2 -11502.167} C_VEL
LIN {X 0,Y 390.138,Z 390.381,A -85,B 0,C 180,E1 -11505.392,E2 -11505.392} C_VEL
LIN {X 0,Y 390.151,Z 390.387,A -85,B 0,C 180,E1 -11508.571,E2 -11508.571} C_VEL
LIN {X 0,Y 390.335,Z 390.361,A -85,B 0,C 180,E1 -11511.993,E2 -11511.993} C_VEL
LIN {X 0,Y 390.221,Z 390.372,A -85,B 0,C 180,E1 -11514.834,E2 -11514.834} C_VEL
LIN {X 0,Y 390.414,Z 390.349,A -85,B 0,C 180,E1 -11517.937,E2 -11517.937} C_VEL
LIN {X 0,Y 390.543,Z 390.331,A -85,B 0,C 180,E1 -11520,E2 -11520} C_VEL
LIN {X 0,Y 390.309,Z 390.359,A -85,B 0,C 180,E1 -11523.097,E2 -11523.097} C_VEL
LIN {X 0,Y 390.323,Z 390.363,A -85,B 0,C 180,E1 -11526.202,E2 -11526.202} C_VEL
LIN {X 0,Y 390.307,Z 390.362,A -85,B 0,C 180,E1 -11528.282,E2 -11528.282} C_VEL
LIN {X 0,Y 390.17,Z 390.383,A -85,B 0,C 180,E1 -11532.483,E2 -11532.483} C_VEL
LIN {X 0,Y 390.131,Z 390.386,A -85,B 0,C 180,E1 -11535.677,E2 -11535.677} C_VEL
LIN {X 0,Y 390.098,Z 390.389,A -85,B 0,C 180,E1 -11538.923,E2 -11538.923} C_VEL
LIN {X 0,Y 390.033,Z 390.397,A -85,B 0,C 180,E1 -11542.235,E2 -11542.235} C_VEL
LIN {X 0,Y 390.112,Z 390.387,A -85,B 0,C 180,E1 -11545.744,E2 -11545.744} C_VEL
LIN {X 0,Y 390.052,Z 390.397,A -85,B 0,C 180,E1 -11549.11,E2 -11549.11} C_VEL
LIN {X 0,Y 390.036,Z 390.402,A -85,B 0,C 180,E1 -11552.722,E2 -11552.722} C_VEL
LIN {X 0,Y 390.052,Z 390.397,A -85,B 0,C 180,E1 -11555.826,E2 -11555.826} C_VEL
LIN {X 0,Y 390.069,Z 390.394,A -85,B 0,C 180,E1 -11559.22,E2 -11559.22} C_VEL
LIN {X 0,Y 390.116,Z 390.377,A -85,B 0,C 180,E1 -11562.388,E2 -11562.388} C_VEL
LIN {X 0,Y 390.059,Z 390.391,A -85,B 0,C 180,E1 -11565.358,E2 -11565.358} C_VEL
LIN {X 0,Y 390.067,Z 390.392,A -85,B 0,C 180,E1 -11569.177,E2 -11569.177} C_VEL
LIN {X 0,Y 390.043,Z 390.399,A -85,B 0,C 180,E1 -11572.45,E2 -11572.45} C_VEL
LIN {X 0,Y 390.066,Z 390.393,A -85,B 0,C 180,E1 -11575.976,E2 -11575.976} C_VEL
LIN {X 0,Y 390.046,Z 390.399,A -85,B 0,C 180,E1 -11579.87,E2 -11579.87} C_VEL
LIN {X 0,Y 390.133,Z 390.595,A -85,B 0,C 180,E1 -11581.388,E2 -11581.388} C_VEL
LIN {X 0,Y 392.047,Z 399.004,A -85,B 0,C 180,E1 -11583.679,E2 -11583.679} C_VEL
LIN {X 0,Y 393.744,Z 408.24,A -85,B 0,C 180,E1 -11586.043,E2 -11586.043} C_VEL
LIN {X 0,Y 393.295,Z 415.293,A -85,B 0,C 180,E1 -11587.684,E2 -11587.684} C_VEL
LIN {X 0,Y 392.823,Z 420.906,A -85,B 0,C 180,E1 -11588.932,E2 -11588.932} C_VEL
LIN {X 0,Y 393.705,Z 425.403,A -85,B 0,C 180,E1 -11589.133,E2 -11589.133} C_VEL
LIN {X 0,Y 397.656,Z 445.647,A -85,B 0,C 180,E1 -11589.778,E2 -11589.778} C_VEL
LIN {X 0,Y 398.143,Z 450.948,A -85,B 0,C 180,E1 -11589.91,E2 -11589.91} C_VEL
LIN {X 0,Y 396.876,Z 529.392,A -85,B 0,C 180,E1 -11591.383,E2 -11591.383} C_VEL
LIN {X 0,Y 396.252,Z 543.014,A -85,B 0,C 180,E1 -11591.852,E2 -11591.852} C_VEL
LIN {X 0,Y 395.472,Z 555.358,A -85,B 0,C 180,E1 -11592.483,E2 -11592.483} C_VEL
LIN {X 0,Y 394.519,Z 567.185,A -85,B 0,C 180,E1 -11593.307,E2 -11593.307} C_VEL
LIN {X 0,Y 393.482,Z 578.55,A -85,B 0,C 180,E1 -11594.327,E2 -11594.327} C_VEL
LIN {X 0,Y 392.454,Z 588.815,A -85,B 0,C 180,E1 -11595.481,E2 -11595.481} C_VEL
LIN {X 0,Y 391.639,Z 598.048,A -85,B 0,C 180,E1 -11596.774,E2 -11596.774} C_VEL
LIN {X 0,Y 390.552,Z 607.022,A -85,B 0,C 180,E1 -11598.321,E2 -11598.321} C_VEL
LIN {X 0,Y 389.879,Z 614.263,A -85,B 0,C 180,E1 -11599.878,E2 -11599.878} C_VEL
LIN {X 0,Y 389.26,Z 620.905,A -85,B 0,C 180,E1 -11601.696,E2 -11601.696} C_VEL
LIN {X 0,Y 388.922,Z 625.307,A -85,B 0,C 180,E1 -11603.255,E2 -11603.255} C_VEL
LIN {X 0,Y 388.803,Z 628.647,A -85,B 0,C 180,E1 -11604.815,E2 -11604.815} C_VEL
LIN {X 0,Y 388.7,Z 630.314,A -85,B 0,C 180,E1 -11605.853,E2 -11605.853} C_VEL
LIN {X 0,Y 388.617,Z 632.457,A -85,B 0,C 180,E1 -11607.927,E2 -11607.927} C_VEL
LIN {X 0,Y 388.655,Z 632.9,A -85,B 0,C 180,E1 -11608.964,E2 -11608.964} C_VEL
LIN {X 0,Y 388.672,Z 632.95,A -85,B 0,C 180,E1 -11610,E2 -11610} C_VEL
LIN {X 0,Y 388.655,Z 632.615,A -85,B 0,C 180,E1 -11611.036,E2 -11611.036} C_VEL
LIN {X 0,Y 388.618,Z 631.894,A -85,B 0,C 180,E1 -11612.073,E2 -11612.073} C_VEL
LIN {X 0,Y 388.602,Z 630.735,A -85,B 0,C 180,E1 -11613.11,E2 -11613.11} C_VEL
LIN {X 0,Y 388.694,Z 629.157,A -85,B 0,C 180,E1 -11614.148,E2 -11614.148} C_VEL
LIN {X 0,Y 388.741,Z 625.812,A -85,B 0,C 180,E1 -11615.775,E2 -11615.775} C_VEL
LIN {X 0,Y 388.96,Z 621.723,A -85,B 0,C 180,E1 -11617.266,E2 -11617.266} C_VEL
LIN {X 0,Y 389.392,Z 615.262,A -85,B 0,C 180,E1 -11619.087,E2 -11619.087} C_VEL
LIN {X 0,Y 389.871,Z 608.172,A -85,B 0,C 180,E1 -11620.648,E2 -11620.648} C_VEL
LIN {X 0,Y 390.601,Z 599.297,A -85,B 0,C 180,E1 -11622.205,E2 -11622.205} C_VEL
LIN {X 0,Y 391.316,Z 590.186,A -85,B 0,C 180,E1 -11623.502,E2 -11623.502} C_VEL
LIN {X 0,Y 392.084,Z 580.12,A -85,B 0,C 180,E1 -11624.666,E2 -11624.666} C_VEL
LIN {X 0,Y 392.87,Z 568.902,A -85,B 0,C 180,E1 -11625.698,E2 -11625.698} C_VEL
LIN {X 0,Y 393.758,Z 556.316,A -85,B 0,C 180,E1 -11626.593,E2 -11626.593} C_VEL
LIN {X 0,Y 394.394,Z 543.388,A -85,B 0,C 180,E1 -11627.266,E2 -11627.266} C_VEL
LIN {X 0,Y 394.933,Z 529.555,A -85,B 0,C 180,E1 -11627.743,E2 -11627.743} C_VEL
LIN {X 0,Y 395.903,Z 447.66,A -85,B 0,C 180,E1 -11629.259,E2 -11629.259} C_VEL
LIN {X 0,Y 391.816,Z 421.452,A -85,B 0,C 180,E1 -11629.943,E2 -11629.943} C_VEL
LIN {X 0,Y 391.913,Z 418.663,A -85,B 0,C 180,E1 -11630.468,E2 -11630.468} C_VEL
LIN {X 0,Y 392.88,Z 406.485,A -85,B 0,C 180,E1 -11633.175,E2 -11633.175} C_VEL
LIN {X 0,Y 392.276,Z 401.548,A -85,B 0,C 180,E1 -11634.334,E2 -11634.334} C_VEL
LIN {X 0,Y 390.154,Z 390.454,A -85,B 0,C 180,E1 -11637.09,E2 -11637.09} C_VEL
LIN {X 0,Y 390.04,Z 390.398,A -85,B 0,C 180,E1 -11640.299,E2 -11640.299} C_VEL
LIN {X 0,Y 390.068,Z 390.395,A -85,B 0,C 180,E1 -11644.024,E2 -11644.024} C_VEL
LIN {X 0,Y 390.046,Z 390.402,A -85,B 0,C 180,E1 -11647.551,E2 -11647.551} C_VEL
LIN {X 0,Y 390.057,Z 390.395,A -85,B 0,C 180,E1 -11650.821,E2 -11650.821} C_VEL
LIN {X 0,Y 390.06,Z 390.397,A -85,B 0,C 180,E1 -11653.887,E2 -11653.887} C_VEL
LIN {X 0,Y 390.112,Z 390.388,A -85,B 0,C 180,E1 -11656.797,E2 -11656.797} C_VEL
LIN {X 0,Y 390.076,Z 390.397,A -85,B 0,C 180,E1 -11659.563,E2 -11659.563} C_VEL
LIN {X 0,Y 390.045,Z 390.396,A -85,B 0,C 180,E1 -11662.448,E2 -11662.448} C_VEL
LIN {X 0,Y 390.065,Z 390.395,A -85,B 0,C 180,E1 -11666.045,E2 -11666.045} C_VEL
LIN {X 0,Y 390.043,Z 390.399,A -85,B 0,C 180,E1 -11669.869,E2 -11669.869} C_VEL
LIN {X 0,Y 390.109,Z 390.393,A -85,B 0,C 180,E1 -11673.231,E2 -11673.231} C_VEL
LIN {X 0,Y 390.072,Z 390.394,A -85,B 0,C 180,E1 -11676.76,E2 -11676.76} C_VEL
LIN {X 0,Y 390.099,Z 390.391,A -85,B 0,C 180,E1 -11679.983,E2 -11679.983} C_VEL
LIN {X 0,Y 390.133,Z 390.391,A -85,B 0,C 180,E1 -11683.248,E2 -11683.248} C_VEL
LIN {X 0,Y 390.189,Z 390.379,A -85,B 0,C 180,E1 -11686.561,E2 -11686.561} C_VEL
LIN {X 0,Y 390.199,Z 390.378,A -85,B 0,C 180,E1 -11690.671,E2 -11690.671} C_VEL
LIN {X 0,Y 390.322,Z 390.364,A -85,B 0,C 180,E1 -11693.798,E2 -11693.798} C_VEL
LIN {X 0,Y 390.415,Z 390.352,A -85,B 0,C 180,E1 -11697.937,E2 -11697.937} C_VEL
LIN {X 0,Y 390.544,Z 390.335,A -85,B 0,C 180,E1 -11700,E2 -11700} C_VEL
LIN {X 0,Y 390.311,Z 390.368,A -85,B 0,C 180,E1 -11703.096,E2 -11703.096} C_VEL
LIN {X 0,Y 390.298,Z 390.365,A -85,B 0,C 180,E1 -11706.648,E2 -11706.648} C_VEL
LIN {X 0,Y 390.199,Z 390.382,A -85,B 0,C 180,E1 -11709.329,E2 -11709.329} C_VEL
LIN {X 0,Y 390.189,Z 390.383,A -85,B 0,C 180,E1 -11713.439,E2 -11713.439} C_VEL
LIN {X 0,Y 390.143,Z 390.389,A -85,B 0,C 180,E1 -11717.308,E2 -11717.308} C_VEL
LIN {X 0,Y 390.082,Z 390.393,A -85,B 0,C 180,E1 -11720.47,E2 -11720.47} C_VEL
LIN {X 0,Y 390.085,Z 390.397,A -85,B 0,C 180,E1 -11723.351,E2 -11723.351} C_VEL
LIN {X 0,Y 390.109,Z 390.391,A -85,B 0,C 180,E1 -11726.768,E2 -11726.768} C_VEL
LIN {X 0,Y 390.04,Z 390.397,A -85,B 0,C 180,E1 -11730.3,E2 -11730.3} C_VEL
LIN {X 0,Y 390.064,Z 390.394,A -85,B 0,C 180,E1 -11734.025,E2 -11734.025} C_VEL
LIN {X 0,Y 390.042,Z 390.399,A -85,B 0,C 180,E1 -11737.552,E2 -11737.552} C_VEL
LIN {X 0,Y 390.054,Z 390.399,A -85,B 0,C 180,E1 -11740.822,E2 -11740.822} C_VEL
LIN {X 0,Y 390.054,Z 390.396,A -85,B 0,C 180,E1 -11743.887,E2 -11743.887} C_VEL
LIN {X 0,Y 390.078,Z 390.394,A -85,B 0,C 180,E1 -11747.62,E2 -11747.62} C_VEL
LIN {X 0,Y 390.094,Z 390.395,A -85,B 0,C 180,E1 -11750.909,E2 -11750.909} C_VEL
LIN {X 0,Y 390.085,Z 390.395,A -85,B 0,C 180,E1 -11754.794,E2 -11754.794} C_VEL
LIN {X 0,Y 390.023,Z 390.401,A -85,B 0,C 180,E1 -11758.496,E2 -11758.496} C_VEL
LIN {X 0,Y 390.117,Z 390.387,A -85,B 0,C 180,E1 -11762.07,E2 -11762.07} C_VEL
LIN {X 0,Y 390.08,Z 390.393,A -85,B 0,C 180,E1 -11765.52,E2 -11765.52} C_VEL
LIN {X 0,Y 390.056,Z 390.4,A -85,B 0,C 180,E1 -11768.878,E2 -11768.878} C_VEL
LIN {X 0,Y 390.129,Z 390.386,A -85,B 0,C 180,E1 -11772.167,E2 -11772.167} C_VEL
LIN {X 0,Y 390.145,Z 390.389,A -85,B 0,C 180,E1 -11775.393,E2 -11775.393} C_VEL
LIN {X 0,Y 390.207,Z 390.508,A -85,B 0,C 180,E1 -11777.98,E2 -11777.98} C_VEL
LIN {X 0,Y 392.312,Z 402.061,A -85,B 0,C 180,E1 -11780.982,E2 -11780.982} C_VEL
LIN {X 0,Y 391.874,Z 408.515,A -85,B 0,C 180,E1 -11782.529,E2 -11782.529} C_VEL
LIN {X 0,Y 391.816,Z 411.264,A -85,B 0,C 180,E1 -11783.107,E2 -11783.107} C_VEL
LIN {X 0,Y 393.848,Z 422.245,A -85,B 0,C 180,E1 -11783.428,E2 -11783.428} C_VEL
LIN {X 0,Y 396.139,Z 435.995,A -85,B 0,C 180,E1 -11783.784,E2 -11783.784} C_VEL
LIN {X 0,Y 394.983,Z 518.266,A -85,B 0,C 180,E1 -11785.295,E2 -11785.295} C_VEL
LIN {X 0,Y 394.536,Z 531.623,A -85,B 0,C 180,E1 -11785.748,E2 -11785.748} C_VEL
LIN {X 0,Y 393.969,Z 543.756,A -85,B 0,C 180,E1 -11786.356,E2 -11786.356} C_VEL
LIN {X 0,Y 393.23,Z 555.899,A -85,B 0,C 180,E1 -11787.183,E2 -11787.183} C_VEL
LIN {X 0,Y 392.327,Z 567.433,A -85,B 0,C 180,E1 -11788.203,E2 -11788.203} C_VEL
LIN {X 0,Y 391.532,Z 577.8,A -85,B 0,C 180,E1 -11789.357,E2 -11789.357} C_VEL
LIN {X 0,Y 390.868,Z 586.281,A -85,B 0,C 180,E1 -11790.515,E2 -11790.515} C_VEL
LIN {X 0,Y 390.177,Z 594.12,A -85,B 0,C 180,E1 -11791.806,E2 -11791.806} C_VEL
LIN {X 0,Y 389.668,Z 601.76,A -85,B 0,C 180,E1 -11793.36,E2 -11793.36} C_VEL
LIN {X 0,Y 389.17,Z 607.02,A -85,B 0,C 180,E1 -11794.661,E2 -11794.661} C_VEL
LIN {X 0,Y 388.988,Z 612.655,A -85,B 0,C 180,E1 -11796.431,E2 -11796.431} C_VEL
LIN {X 0,Y 388.801,Z 616.078,A -85,B 0,C 180,E1 -11797.814,E2 -11797.814} C_VEL
LIN {X 0,Y 388.011,Z 617.742,A -85,B 0,C 180,E1 -11798.644,E2 -11798.644} C_VEL
LIN {X 0,Y 385.023,Z 619.9,A -85,B 0,C 180,E1 -11800.01,E2 -11800.01} C_VEL
LIN {X 0,Y 382.574,Z 621.097,A -85,B 0,C 180,E1 -11801.128,E2 -11801.128} C_VEL
LIN {X 0,Y 381.552,Z 621.706,A -85,B 0,C 180,E1 -11802,E2 -11802} C_VEL
LIN {X 0,Y 381.481,Z 621.836,A -85,B 0,C 180,E1 -11802.296,E2 -11802.296} C_VEL
LIN {X 0,Y 381.362,Z 622.076,A -85,B 0,C 180,E1 -11803.861,E2 -11803.861} C_VEL
LIN {X 0,Y 381.377,Z 621.733,A -85,B 0,C 180,E1 -11804.95,E2 -11804.95} C_VEL
LIN {X 0,Y 381.513,Z 620.313,A -85,B 0,C 180,E1 -11806.682,E2 -11806.682} C_VEL
LIN {X 0,Y 381.813,Z 617.098,A -85,B 0,C 180,E1 -11808.791,E2 -11808.791} C_VEL
LIN {X 0,Y 382.137,Z 613.34,A -85,B 0,C 180,E1 -11810.452,E2 -11810.452} C_VEL
LIN {X 0,Y 382.632,Z 608.361,A -85,B 0,C 180,E1 -11812.118,E2 -11812.118} C_VEL
LIN {X 0,Y 383.304,Z 601.997,A -85,B 0,C 180,E1 -11813.789,E2 -11813.789} C_VEL
LIN {X 0,Y 384.194,Z 593.967,A -85,B 0,C 180,E1 -11815.459,E2 -11815.459} C_VEL
LIN {X 0,Y 385.192,Z 584.982,A -85,B 0,C 180,E1 -11816.946,E2 -11816.946} C_VEL
LIN {X 0,Y 386.221,Z 575.368,A -85,B 0,C 180,E1 -11818.236,E2 -11818.236} C_VEL
LIN {X 0,Y 387.314,Z 565.22,A -85,B 0,C 180,E1 -11819.335,E2 -11819.335} C_VEL
LIN {X 0,Y 388.257,Z 554.209,A -85,B 0,C 180,E1 -11820.287,E2 -11820.287} C_VEL
LIN {X 0,Y 389.156,Z 542.776,A -85,B 0,C 180,E1 -11821.052,E2 -11821.052} C_VEL
LIN {X 0,Y 389.904,Z 529.806,A -85,B 0,C 180,E1 -11821.692,E2 -11821.692} C_VEL
LIN {X 0,Y 390.441,Z 517.607,A -85,B 0,C 180,E1 -11822.087,E2 -11822.087} C_VEL
LIN {X 0,Y 391.75,Z 436.366,A -85,B 0,C 180,E1 -11823.626,E2 -11823.626} C_VEL
LIN {X 0,Y 387.365,Z 416.057,A -85,B 0,C 180,E1 -11824.325,E2 -11824.325} C_VEL
LIN {X 0,Y 386.294,Z 411.37,A -85,B 0,C 180,E1 -11824.536,E2 -11824.536} C_VEL
LIN {X 0,Y 386.304,Z 407.001,A -85,B 0,C 180,E1 -11825.602,E2 -11825.602} C_VEL
LIN {X 0,Y 383.838,Z 394.771,A -85,B 0,C 180,E1 -11829.054,E2 -11829.054} C_VEL
LIN {X 0,Y 383.062,Z 391.311,A -85,B 0,C 180,E1 -11830.143,E2 -11830.143} C_VEL
LIN {X 0,Y 383.061,Z 391.267,A -85,B 0,C 180,E1 -11832.788,E2 -11832.788} C_VEL
LIN {X 0,Y 383.065,Z 391.267,A -85,B 0,C 180,E1 -11835.799,E2 -11835.799} C_VEL
LIN {X 0,Y 383.039,Z 391.268,A -85,B 0,C 180,E1 -11838.785,E2 -11838.785} C_VEL
LIN {X 0,Y 382.998,Z 391.273,A -85,B 0,C 180,E1 -11842.095,E2 -11842.095} C_VEL
LIN {X 0,Y 383.012,Z 391.264,A -85,B 0,C 180,E1 -11845.331,E2 -11845.331} C_VEL
LIN {X 0,Y 383.031,Z 391.272,A -85,B 0,C 180,E1 -11847.852,E2 -11847.852} C_VEL
LIN {X 0,Y 383.056,Z 391.267,A -85,B 0,C 180,E1 -11851.72,E2 -11851.72} C_VEL
LIN {X 0,Y 383.045,Z 391.27,A -85,B 0,C 180,E1 -11855.039,E2 -11855.039} C_VEL
LIN {X 0,Y 383.011,Z 391.27,A -85,B 0,C 180,E1 -11858.47,E2 -11858.47} C_VEL
LIN {X 0,Y 383.086,Z 391.259,A -85,B 0,C 180,E1 -11861.828,E2 -11861.828} C_VEL
LIN {X 0,Y 383.103,Z 391.259,A -85,B 0,C 180,E1 -11865.118,E2 -11865.118} C_VEL
LIN {X 0,Y 383.1,Z 391.264,A -85,B 0,C 180,E1 -11868.358,E2 -11868.358} C_VEL
LIN {X 0,Y 383.295,Z 391.238,A -85,B 0,C 180,E1 -11871.933,E2 -11871.933} C_VEL
LIN {X 0,Y 383.193,Z 391.246,A -85,B 0,C 180,E1 -11874.738,E2 -11874.738} C_VEL
LIN {X 0,Y 383.383,Z 391.225,A -85,B 0,C 180,E1 -11877.899,E2 -11877.899} C_VEL
LIN {X 0,Y 383.513,Z 391.206,A -85,B 0,C 180,E1 -11880,E2 -11880} C_VEL
LIN {X 0,Y 383.245,Z 391.238,A -85,B 0,C 180,E1 -11883.154,E2 -11883.154} C_VEL
LIN {X 0,Y 383.28,Z 391.241,A -85,B 0,C 180,E1 -11886.317,E2 -11886.317} C_VEL
LIN {X 0,Y 383.252,Z 391.24,A -85,B 0,C 180,E1 -11888.436,E2 -11888.436} C_VEL
LIN {X 0,Y 383.099,Z 391.262,A -85,B 0,C 180,E1 -11891.642,E2 -11891.642} C_VEL
LIN {X 0,Y 383.104,Z 391.262,A -85,B 0,C 180,E1 -11894.882,E2 -11894.882} C_VEL
LIN {X 0,Y 383.081,Z 391.26,A -85,B 0,C 180,E1 -11898.173,E2 -11898.173} C_VEL
LIN {X 0,Y 382.989,Z 391.273,A -85,B 0,C 180,E1 -11901.531,E2 -11901.531} C_VEL
LIN {X 0,Y 383.045,Z 391.271,A -85,B 0,C 180,E1 -11904.961,E2 -11904.961} C_VEL
LIN {X 0,Y 383.034,Z 391.273,A -85,B 0,C 180,E1 -11908.493,E2 -11908.493} C_VEL
LIN {X 0,Y 383.003,Z 391.275,A -85,B 0,C 180,E1 -11912.151,E2 -11912.151} C_VEL
LIN {X 0,Y 383.012,Z 391.274,A -85,B 0,C 180,E1 -11914.669,E2 -11914.669} C_VEL
LIN {X 0,Y 382.998,Z 391.273,A -85,B 0,C 180,E1 -11917.905,E2 -11917.905} C_VEL
LIN {X 0,Y 383.042,Z 391.253,A -85,B 0,C 180,E1 -11921.34,E2 -11921.34} C_VEL
LIN {X 0,Y 383.031,Z 391.275,A -85,B 0,C 180,E1 -11924.31,E2 -11924.31} C_VEL
LIN {X 0,Y 383.006,Z 391.272,A -85,B 0,C 180,E1 -11927.241,E2 -11927.241} C_VEL
LIN {X 0,Y 383.015,Z 391.268,A -85,B 0,C 180,E1 -11930.414,E2 -11930.414} C_VEL
LIN {X 0,Y 383.024,Z 391.269,A -85,B 0,C 180,E1 -11934.046,E2 -11934.046} C_VEL
LIN {X 0,Y 382.985,Z 391.28,A -85,B 0,C 180,E1 -11937.579,E2 -11937.579} C_VEL
LIN {X 0,Y 383.052,Z 391.357,A -85,B 0,C 180,E1 -11940.909,E2 -11940.909} C_VEL
LIN {X 0,Y 384.914,Z 399.508,A -85,B 0,C 180,E1 -11943.22,E2 -11943.22} C_VEL
LIN {X 0,Y 386.874,Z 409.719,A -85,B 0,C 180,E1 -11945.902,E2 -11945.902} C_VEL
LIN {X 0,Y 386.395,Z 416.663,A -85,B 0,C 180,E1 -11947.546,E2 -11947.546} C_VEL
LIN {X 0,Y 385.996,Z 420.772,A -85,B 0,C 180,E1 -11948.473,E2 -11948.473} C_VEL
LIN {X 0,Y 386.828,Z 424.721,A -85,B 0,C 180,E1 -11948.664,E2 -11948.664} C_VEL
LIN {X 0,Y 391.153,Z 446.6,A -85,B 0,C 180,E1 -11949.389,E2 -11949.389} C_VEL
LIN {X 0,Y 391.612,Z 451.533,A -85,B 0,C 180,E1 -11949.516,E2 -11949.516} C_VEL
LIN {X 0,Y 390.292,Z 529.115,A -85,B 0,C 180,E1 -11950.992,E2 -11950.992} C_VEL
LIN {X 0,Y 389.653,Z 542.709,A -85,B 0,C 180,E1 -11951.465,E2 -11951.465} C_VEL
LIN {X 0,Y 388.803,Z 555.106,A -85,B 0,C 180,E1 -11952.105,E2 -11952.105} C_VEL
LIN {X 0,Y 387.92,Z 566.175,A -85,B 0,C 180,E1 -11952.879,E2 -11952.879} C_VEL
LIN {X 0,Y 386.79,Z 577.699,A -85,B 0,C 180,E1 -11953.914,E2 -11953.914} C_VEL
LIN {X 0,Y 385.757,Z 587.711,A -85,B 0,C 180,E1 -11955.04,E2 -11955.04} C_VEL
LIN {X 0,Y 384.875,Z 596.597,A -85,B 0,C 180,E1 -11956.268,E2 -11956.268} C_VEL
LIN {X 0,Y 383.912,Z 604.462,A -85,B 0,C 180,E1 -11957.579,E2 -11957.579} C_VEL
LIN {X 0,Y 383.117,Z 612.166,A -85,B 0,C 180,E1 -11959.163,E2 -11959.163} C_VEL
LIN {X 0,Y 382.395,Z 619.261,A -85,B 0,C 180,E1 -11961.013,E2 -11961.013} C_VEL
LIN {X 0,Y 381.959,Z 624.003,A -85,B 0,C 180,E1 -11962.6,E2 -11962.6} C_VEL
LIN {X 0,Y 381.752,Z 626.846,A -85,B 0,C 180,E1 -11963.792,E2 -11963.792} C_VEL
LIN {X 0,Y 381.63,Z 630.287,A -85,B 0,C 180,E1 -11965.776,E2 -11965.776} C_VEL
LIN {X 0,Y 381.514,Z 632.388,A -85,B 0,C 180,E1 -11967.889,E2 -11967.889} C_VEL
LIN {X 0,Y 381.554,Z 632.807,A -85,B 0,C 180,E1 -11968.945,E2 -11968.945} C_VEL
LIN {X 0,Y 381.587,Z 632.841,A -85,B 0,C 180,E1 -11970,E2 -11970} C_VEL
LIN {X 0,Y 381.554,Z 632.491,A -85,B 0,C 180,E1 -11971.056,E2 -11971.056} C_VEL
LIN {X 0,Y 381.516,Z 631.749,A -85,B 0,C 180,E1 -11972.112,E2 -11972.112} C_VEL
LIN {X 0,Y 381.516,Z 630.563,A -85,B 0,C 180,E1 -11973.168,E2 -11973.168} C_VEL
LIN {X 0,Y 381.629,Z 628.024,A -85,B 0,C 180,E1 -11974.754,E2 -11974.754} C_VEL
LIN {X 0,Y 381.712,Z 624.462,A -85,B 0,C 180,E1 -11976.343,E2 -11976.343} C_VEL
LIN {X 0,Y 382.018,Z 619.785,A -85,B 0,C 180,E1 -11977.931,E2 -11977.931} C_VEL
LIN {X 0,Y 382.503,Z 612.718,A -85,B 0,C 180,E1 -11979.785,E2 -11979.785} C_VEL
LIN {X 0,Y 383.07,Z 605.047,A -85,B 0,C 180,E1 -11981.375,E2 -11981.375} C_VEL
LIN {X 0,Y 383.786,Z 597.186,A -85,B 0,C 180,E1 -11982.694,E2 -11982.694} C_VEL
LIN {X 0,Y 384.658,Z 586.666,A -85,B 0,C 180,E1 -11984.122,E2 -11984.122} C_VEL
LIN {X 0,Y 385.482,Z 575.558,A -85,B 0,C 180,E1 -11985.329,E2 -11985.329} C_VEL
LIN {X 0,Y 386.2,Z 564.845,A -85,B 0,C 180,E1 -11986.248,E2 -11986.248} C_VEL
LIN {X 0,Y 387.088,Z 551.946,A -85,B 0,C 180,E1 -11987.092,E2 -11987.092} C_VEL
LIN {X 0,Y 387.759,Z 538.865,A -85,B 0,C 180,E1 -11987.707,E2 -11987.707} C_VEL
LIN {X 0,Y 388.14,Z 525.788,A -85,B 0,C 180,E1 -11988.098,E2 -11988.098} C_VEL
LIN {X 0,Y 389.11,Z 448.6,A -85,B 0,C 180,E1 -11989.532,E2 -11989.532} C_VEL
LIN {X 0,Y 384.876,Z 421.247,A -85,B 0,C 180,E1 -11990.264,E2 -11990.264} C_VEL
LIN {X 0,Y 385.103,Z 417.087,A -85,B 0,C 180,E1 -11991.126,E2 -11991.126} C_VEL
LIN {X 0,Y 385.855,Z 406.112,A -85,B 0,C 180,E1 -11993.622,E2 -11993.622} C_VEL
LIN {X 0,Y 383.581,Z 393.628,A -85,B 0,C 180,E1 -11996.683,E2 -11996.683} C_VEL
LIN {X 0,Y 383.121,Z 391.309,A -85,B 0,C 180,E1 -11997.333,E2 -11997.333} C_VEL
LIN {X 0,Y 382.984,Z 391.28,A -85,B 0,C 180,E1 -12000.918,E2 -12000.918} C_VEL
LIN {X 0,Y 383.018,Z 391.271,A -85,B 0,C 180,E1 -12004.667,E2 -12004.667} C_VEL
LIN {X 0,Y 383.002,Z 391.276,A -85,B 0,C 180,E1 -12007.904,E2 -12007.904} C_VEL
LIN {X 0,Y 382.985,Z 391.28,A -85,B 0,C 180,E1 -12011.347,E2 -12011.347} C_VEL
LIN {X 0,Y 383.008,Z 391.273,A -85,B 0,C 180,E1 -12014.305,E2 -12014.305} C_VEL
LIN {X 0,Y 383.073,Z 391.269,A -85,B 0,C 180,E1 -12017.249,E2 -12017.249} C_VEL
LIN {X 0,Y 383.02,Z 391.271,A -85,B 0,C 180,E1 -12020.412,E2 -12020.412} C_VEL
LIN {X 0,Y 383.024,Z 391.272,A -85,B 0,C 180,E1 -12024.044,E2 -12024.044} C_VEL
LIN {X 0,Y 382.983,Z 391.28,A -85,B 0,C 180,E1 -12027.578,E2 -12027.578} C_VEL
LIN {X 0,Y 382.988,Z 391.275,A -85,B 0,C 180,E1 -12030.3,E2 -12030.3} C_VEL
LIN {X 0,Y 383.053,Z 391.268,A -85,B 0,C 180,E1 -12032.698,E2 -12032.698} C_VEL
LIN {X 0,Y 383.047,Z 391.271,A -85,B 0,C 180,E1 -12035.039,E2 -12035.039} C_VEL
LIN {X 0,Y 382.988,Z 391.275,A -85,B 0,C 180,E1 -12038.469,E2 -12038.469} C_VEL
LIN {X 0,Y 383.085,Z 391.266,A -85,B 0,C 180,E1 -12041.827,E2 -12041.827} C_VEL
LIN {X 0,Y 383.105,Z 391.265,A -85,B 0,C 180,E1 -12045.118,E2 -12045.118} C_VEL
LIN {X 0,Y 383.091,Z 391.263,A -85,B 0,C 180,E1 -12048.358,E2 -12048.358} C_VEL
LIN {X 0,Y 383.259,Z 391.243,A -85,B 0,C 180,E1 -12051.975,E2 -12051.975} C_VEL
LIN {X 0,Y 383.193,Z 391.251,A -85,B 0,C 180,E1 -12054.738,E2 -12054.738} C_VEL
LIN {X 0,Y 383.382,Z 391.228,A -85,B 0,C 180,E1 -12057.899,E2 -12057.899} C_VEL
LIN {X 0,Y 383.514,Z 391.211,A -85,B 0,C 180,E1 -12060,E2 -12060} C_VEL
LIN {X 0,Y 383.247,Z 391.248,A -85,B 0,C 180,E1 -12063.154,E2 -12063.154} C_VEL
LIN {X 0,Y 383.257,Z 391.242,A -85,B 0,C 180,E1 -12066.64,E2 -12066.64} C_VEL
LIN {X 0,Y 383.146,Z 391.26,A -85,B 0,C 180,E1 -12069.502,E2 -12069.502} C_VEL
LIN {X 0,Y 383.12,Z 391.262,A -85,B 0,C 180,E1 -12073.536,E2 -12073.536} C_VEL
LIN {X 0,Y 383.09,Z 391.267,A -85,B 0,C 180,E1 -12077.455,E2 -12077.455} C_VEL
LIN {X 0,Y 383.024,Z 391.273,A -85,B 0,C 180,E1 -12080.647,E2 -12080.647} C_VEL
LIN {X 0,Y 383.029,Z 391.271,A -85,B 0,C 180,E1 -12083.808,E2 -12083.808} C_VEL
LIN {X 0,Y 383.075,Z 391.265,A -85,B 0,C 180,E1 -12086.124,E2 -12086.124} C_VEL
LIN {X 0,Y 383.045,Z 391.269,A -85,B 0,C 180,E1 -12088.492,E2 -12088.492} C_VEL
LIN {X 0,Y 383.008,Z 391.273,A -85,B 0,C 180,E1 -12092.15,E2 -12092.15} C_VEL
LIN {X 0,Y 383.014,Z 391.274,A -85,B 0,C 180,E1 -12094.668,E2 -12094.668} C_VEL
LIN {X 0,Y 382.998,Z 391.274,A -85,B 0,C 180,E1 -12097.904,E2 -12097.904} C_VEL
LIN {X 0,Y 382.982,Z 391.28,A -85,B 0,C 180,E1 -12101.348,E2 -12101.348} C_VEL
LIN {X 0,Y 382.995,Z 391.275,A -85,B 0,C 180,E1 -12104.304,E2 -12104.304} C_VEL
LIN {X 0,Y 383.037,Z 391.274,A -85,B 0,C 180,E1 -12107.245,E2 -12107.245} C_VEL
LIN {X 0,Y 383.02,Z 391.272,A -85,B 0,C 180,E1 -12110.413,E2 -12110.413} C_VEL
LIN {X 0,Y 383.026,Z 391.27,A -85,B 0,C 180,E1 -12114.045,E2 -12114.045} C_VEL
LIN {X 0,Y 382.986,Z 391.277,A -85,B 0,C 180,E1 -12117.578,E2 -12117.578} C_VEL
LIN {X 0,Y 382.992,Z 391.275,A -85,B 0,C 180,E1 -12120.3,E2 -12120.3} C_VEL
LIN {X 0,Y 383.08,Z 391.263,A -85,B 0,C 180,E1 -12124.021,E2 -12124.021} C_VEL
LIN {X 0,Y 383.009,Z 391.275,A -85,B 0,C 180,E1 -12127.335,E2 -12127.335} C_VEL
LIN {X 0,Y 383.062,Z 391.27,A -85,B 0,C 180,E1 -12130.717,E2 -12130.717} C_VEL
LIN {X 0,Y 383.082,Z 391.263,A -85,B 0,C 180,E1 -12134.027,E2 -12134.027} C_VEL
LIN {X 0,Y 383.16,Z 391.325,A -85,B 0,C 180,E1 -12137.722,E2 -12137.722} C_VEL
LIN {X 0,Y 385.275,Z 402.914,A -85,B 0,C 180,E1 -12140.815,E2 -12140.815} C_VEL
LIN {X 0,Y 385.127,Z 408.27,A -85,B 0,C 180,E1 -12142.133,E2 -12142.133} C_VEL
LIN {X 0,Y 384.766,Z 411.244,A -85,B 0,C 180,E1 -12142.781,E2 -12142.781} C_VEL
LIN {X 0,Y 388.734,Z 432.593,A -85,B 0,C 180,E1 -12143.398,E2 -12143.398} C_VEL
LIN {X 0,Y 389.332,Z 436.353,A -85,B 0,C 180,E1 -12143.496,E2 -12143.496} C_VEL
LIN {X 0,Y 388.122,Z 518.753,A -85,B 0,C 180,E1 -12145.04,E2 -12145.04} C_VEL
LIN {X 0,Y 387.643,Z 532.268,A -85,B 0,C 180,E1 -12145.512,E2 -12145.512} C_VEL
LIN {X 0,Y 387.026,Z 544.768,A -85,B 0,C 180,E1 -12146.16,E2 -12146.16} C_VEL
LIN {X 0,Y 386.272,Z 556.645,A -85,B 0,C 180,E1 -12147.001,E2 -12147.001} C_VEL
LIN {X 0,Y 385.34,Z 568.063,A -85,B 0,C 180,E1 -12148.04,E2 -12148.04} C_VEL
LIN {X 0,Y 384.526,Z 578.335,A -85,B 0,C 180,E1 -12149.214,E2 -12149.214} C_VEL
LIN {X 0,Y 383.766,Z 587.565,A -85,B 0,C 180,E1 -12150.524,E2 -12150.524} C_VEL
LIN {X 0,Y 382.965,Z 596.544,A -85,B 0,C 180,E1 -12152.103,E2 -12152.103} C_VEL
LIN {X 0,Y 382.446,Z 603.773,A -85,B 0,C 180,E1 -12153.687,E2 -12153.687} C_VEL
LIN {X 0,Y 382.063,Z 609.555,A -85,B 0,C 180,E1 -12155.277,E2 -12155.277} C_VEL
LIN {X 0,Y 381.827,Z 613.978,A -85,B 0,C 180,E1 -12156.818,E2 -12156.818} C_VEL
LIN {X 0,Y 381.623,Z 617.581,A -85,B 0,C 180,E1 -12158.472,E2 -12158.472} C_VEL
LIN {X 0,Y 381.497,Z 619.309,A -85,B 0,C 180,E1 -12159.543,E2 -12159.543} C_VEL
LIN {X 0,Y 381.443,Z 620.624,A -85,B 0,C 180,E1 -12160.617,E2 -12160.617} C_VEL
LIN {X 0,Y 381.481,Z 621.836,A -85,B 0,C 180,E1 -12162.296,E2 -12162.296} C_VEL
LIN {X 0,Y 380.827,Z 622.142,A -85,B 0,C 180,E1 -12163.177,E2 -12163.177} C_VEL
LIN {X 0,Y 377.923,Z 622.063,A -85,B 0,C 180,E1 -12164.61,E2 -12164.61} C_VEL
LIN {X 0,Y 375.488,Z 621.428,A -85,B 0,C 180,E1 -12165.764,E2 -12165.764} C_VEL
LIN {X 0,Y 374.494,Z 620.589,A -85,B 0,C 180,E1 -12166.652,E2 -12166.652} C_VEL
LIN {X 0,Y 374.442,Z 620.237,A -85,B 0,C 180,E1 -12166.95,E2 -12166.95} C_VEL
LIN {X 0,Y 374.789,Z 616.807,A -85,B 0,C 180,E1 -12169.156,E2 -12169.156} C_VEL
LIN {X 0,Y 375.161,Z 612.914,A -85,B 0,C 180,E1 -12170.85,E2 -12170.85} C_VEL
LIN {X 0,Y 375.709,Z 607.792,A -85,B 0,C 180,E1 -12172.548,E2 -12172.548} C_VEL
LIN {X 0,Y 376.479,Z 601.272,A -85,B 0,C 180,E1 -12174.247,E2 -12174.247} C_VEL
LIN {X 0,Y 377.445,Z 592.979,A -85,B 0,C 180,E1 -12175.948,E2 -12175.948} C_VEL
LIN {X 0,Y 378.461,Z 584.274,A -85,B 0,C 180,E1 -12177.386,E2 -12177.386} C_VEL
LIN {X 0,Y 379.647,Z 573.876,A -85,B 0,C 180,E1 -12178.77,E2 -12178.77} C_VEL
LIN {X 0,Y 380.818,Z 563.281,A -85,B 0,C 180,E1 -12179.886,E2 -12179.886} C_VEL
LIN {X 0,Y 381.842,Z 551.571,A -85,B 0,C 180,E1 -12180.866,E2 -12180.866} C_VEL
LIN {X 0,Y 382.777,Z 539.574,A -85,B 0,C 180,E1 -12181.628,E2 -12181.628} C_VEL
LIN {X 0,Y 383.519,Z 526.371,A -85,B 0,C 180,E1 -12182.22,E2 -12182.22} C_VEL
LIN {X 0,Y 384.026,Z 512.969,A -85,B 0,C 180,E1 -12182.593,E2 -12182.593} C_VEL
LIN {X 0,Y 385.313,Z 437.663,A -85,B 0,C 180,E1 -12184.027,E2 -12184.027} C_VEL
LIN {X 0,Y 380.693,Z 416.503,A -85,B 0,C 180,E1 -12184.782,E2 -12184.782} C_VEL
LIN {X 0,Y 379.544,Z 411.546,A -85,B 0,C 180,E1 -12185,E2 -12185} C_VEL
LIN {X 0,Y 379.325,Z 408.171,A -85,B 0,C 180,E1 -12185.83,E2 -12185.83} C_VEL
LIN {X 0,Y 377.095,Z 396.992,A -85,B 0,C 180,E1 -12189.051,E2 -12189.051} C_VEL
LIN {X 0,Y 376.012,Z 392.204,A -85,B 0,C 180,E1 -12190.557,E2 -12190.557} C_VEL
LIN {X 0,Y 375.997,Z 392.151,A -85,B 0,C 180,E1 -12193.755,E2 -12193.755} C_VEL
LIN {X 0,Y 375.994,Z 392.152,A -85,B 0,C 180,E1 -12196.799,E2 -12196.799} C_VEL
LIN {X 0,Y 375.994,Z 392.149,A -85,B 0,C 180,E1 -12200.027,E2 -12200.027} C_VEL
LIN {X 0,Y 375.959,Z 392.154,A -85,B 0,C 180,E1 -12203.494,E2 -12203.494} C_VEL
LIN {X 0,Y 375.955,Z 392.145,A -85,B 0,C 180,E1 -12205.888,E2 -12205.888} C_VEL
LIN {X 0,Y 375.963,Z 392.138,A -85,B 0,C 180,E1 -12209.687,E2 -12209.687} C_VEL
LIN {X 0,Y 375.995,Z 392.146,A -85,B 0,C 180,E1 -12212.141,E2 -12212.141} C_VEL
LIN {X 0,Y 375.999,Z 392.147,A -85,B 0,C 180,E1 -12214.538,E2 -12214.538} C_VEL
LIN {X 0,Y 375.973,Z 392.145,A -85,B 0,C 180,E1 -12218.046,E2 -12218.046} C_VEL
LIN {X 0,Y 376.024,Z 392.14,A -85,B 0,C 180,E1 -12221.474,E2 -12221.474} C_VEL
LIN {X 0,Y 376.051,Z 392.139,A -85,B 0,C 180,E1 -12224.832,E2 -12224.832} C_VEL
LIN {X 0,Y 376.051,Z 392.141,A -85,B 0,C 180,E1 -12228.137,E2 -12228.137} C_VEL
LIN {X 0,Y 376.249,Z 392.116,A -85,B 0,C 180,E1 -12231.877,E2 -12231.877} C_VEL
LIN {X 0,Y 376.165,Z 392.121,A -85,B 0,C 180,E1 -12234.64,E2 -12234.64} C_VEL
LIN {X 0,Y 376.35,Z 392.101,A -85,B 0,C 180,E1 -12237.86,E2 -12237.86} C_VEL
LIN {X 0,Y 376.482,Z 392.082,A -85,B 0,C 180,E1 -12240,E2 -12240} C_VEL
LIN {X 0,Y 376.183,Z 392.117,A -85,B 0,C 180,E1 -12243.213,E2 -12243.213} C_VEL
LIN {X 0,Y 376.239,Z 392.119,A -85,B 0,C 180,E1 -12246.435,E2 -12246.435} C_VEL
LIN {X 0,Y 376.198,Z 392.117,A -85,B 0,C 180,E1 -12248.595,E2 -12248.595} C_VEL
LIN {X 0,Y 376.051,Z 392.14,A -85,B 0,C 180,E1 -12251.864,E2 -12251.864} C_VEL
LIN {X 0,Y 376.051,Z 392.142,A -85,B 0,C 180,E1 -12255.168,E2 -12255.168} C_VEL
LIN {X 0,Y 376.016,Z 392.14,A -85,B 0,C 180,E1 -12258.527,E2 -12258.527} C_VEL
LIN {X 0,Y 375.958,Z 392.15,A -85,B 0,C 180,E1 -12261.955,E2 -12261.955} C_VEL
LIN {X 0,Y 375.999,Z 392.145,A -85,B 0,C 180,E1 -12265.462,E2 -12265.462} C_VEL
LIN {X 0,Y 375.964,Z 392.152,A -85,B 0,C 180,E1 -12269.08,E2 -12269.08} C_VEL
LIN {X 0,Y 375.943,Z 392.156,A -85,B 0,C 180,E1 -12272.829,E2 -12272.829} C_VEL
LIN {X 0,Y 375.953,Z 392.153,A -85,B 0,C 180,E1 -12275.416,E2 -12275.416} C_VEL
LIN {X 0,Y 375.973,Z 392.15,A -85,B 0,C 180,E1 -12278.272,E2 -12278.272} C_VEL
LIN {X 0,Y 375.985,Z 392.132,A -85,B 0,C 180,E1 -12281.611,E2 -12281.611} C_VEL
LIN {X 0,Y 375.966,Z 392.147,A -85,B 0,C 180,E1 -12285.263,E2 -12285.263} C_VEL
LIN {X 0,Y 375.948,Z 392.152,A -85,B 0,C 180,E1 -12289.135,E2 -12289.135} C_VEL
LIN {X 0,Y 375.963,Z 392.154,A -85,B 0,C 180,E1 -12291.913,E2 -12291.913} C_VEL
LIN {X 0,Y 375.978,Z 392.151,A -85,B 0,C 180,E1 -12295.334,E2 -12295.334} C_VEL
LIN {X 0,Y 375.956,Z 392.151,A -85,B 0,C 180,E1 -12298.439,E2 -12298.439} C_VEL
LIN {X 0,Y 376,Z 392.369,A -85,B 0,C 180,E1 -12300.541,E2 -12300.541} C_VEL
LIN {X 0,Y 378.13,Z 401.454,A -85,B 0,C 180,E1 -12303.144,E2 -12303.144} C_VEL
LIN {X 0,Y 379.869,Z 410.475,A -85,B 0,C 180,E1 -12305.566,E2 -12305.566} C_VEL
LIN {X 0,Y 379.984,Z 413.326,A -85,B 0,C 180,E1 -12306.28,E2 -12306.28} C_VEL
LIN {X 0,Y 379.22,Z 420.689,A -85,B 0,C 180,E1 -12308.003,E2 -12308.003} C_VEL
LIN {X 0,Y 380.446,Z 426.361,A -85,B 0,C 180,E1 -12308.254,E2 -12308.254} C_VEL
LIN {X 0,Y 384.759,Z 448.117,A -85,B 0,C 180,E1 -12308.997,E2 -12308.997} C_VEL
LIN {X 0,Y 385.114,Z 453.123,A -85,B 0,C 180,E1 -12309.123,E2 -12309.123} C_VEL
LIN {X 0,Y 383.763,Z 528.795,A -85,B 0,C 180,E1 -12310.586,E2 -12310.586} C_VEL
LIN {X 0,Y 383.078,Z 542.477,A -85,B 0,C 180,E1 -12311.066,E2 -12311.066} C_VEL
LIN {X 0,Y 382.2,Z 554.91,A -85,B 0,C 180,E1 -12311.715,E2 -12311.715} C_VEL
LIN {X 0,Y 381.189,Z 566.791,A -85,B 0,C 180,E1 -12312.567,E2 -12312.567} C_VEL
LIN {X 0,Y 380.01,Z 578.185,A -85,B 0,C 180,E1 -12313.619,E2 -12313.619} C_VEL
LIN {X 0,Y 378.891,Z 588.362,A -85,B 0,C 180,E1 -12314.798,E2 -12314.798} C_VEL
LIN {X 0,Y 377.97,Z 596.889,A -85,B 0,C 180,E1 -12316.012,E2 -12316.012} C_VEL
LIN {X 0,Y 376.99,Z 604.678,A -85,B 0,C 180,E1 -12317.347,E2 -12317.347} C_VEL
LIN {X 0,Y 376.152,Z 612.3,A -85,B 0,C 180,E1 -12318.96,E2 -12318.96} C_VEL
LIN {X 0,Y 375.37,Z 619.347,A -85,B 0,C 180,E1 -12320.843,E2 -12320.843} C_VEL
LIN {X 0,Y 374.895,Z 624.05,A -85,B 0,C 180,E1 -12322.46,E2 -12322.46} C_VEL
LIN {X 0,Y 374.675,Z 627.109,A -85,B 0,C 180,E1 -12323.802,E2 -12323.802} C_VEL
LIN {X 0,Y 374.56,Z 630.262,A -85,B 0,C 180,E1 -12325.696,E2 -12325.696} C_VEL
LIN {X 0,Y 374.435,Z 631.495,A -85,B 0,C 180,E1 -12326.772,E2 -12326.772} C_VEL
LIN {X 0,Y 374.414,Z 632.315,A -85,B 0,C 180,E1 -12327.849,E2 -12327.849} C_VEL
LIN {X 0,Y 374.452,Z 632.715,A -85,B 0,C 180,E1 -12328.925,E2 -12328.925} C_VEL
LIN {X 0,Y 374.488,Z 632.732,A -85,B 0,C 180,E1 -12330,E2 -12330} C_VEL
LIN {X 0,Y 374.453,Z 632.365,A -85,B 0,C 180,E1 -12331.076,E2 -12331.076} C_VEL
LIN {X 0,Y 374.416,Z 631.596,A -85,B 0,C 180,E1 -12332.152,E2 -12332.152} C_VEL
LIN {X 0,Y 374.527,Z 628.773,A -85,B 0,C 180,E1 -12334.305,E2 -12334.305} C_VEL
LIN {X 0,Y 374.588,Z 625.169,A -85,B 0,C 180,E1 -12336.074,E2 -12336.074} C_VEL
LIN {X 0,Y 374.841,Z 621.188,A -85,B 0,C 180,E1 -12337.542,E2 -12337.542} C_VEL
LIN {X 0,Y 375.225,Z 615.654,A -85,B 0,C 180,E1 -12339.161,E2 -12339.161} C_VEL
LIN {X 0,Y 375.719,Z 608.728,A -85,B 0,C 180,E1 -12340.781,E2 -12340.781} C_VEL
LIN {X 0,Y 376.507,Z 600.047,A -85,B 0,C 180,E1 -12342.396,E2 -12342.396} C_VEL
LIN {X 0,Y 377.265,Z 591.124,A -85,B 0,C 180,E1 -12343.74,E2 -12343.74} C_VEL
LIN {X 0,Y 378.035,Z 581.619,A -85,B 0,C 180,E1 -12344.912,E2 -12344.912} C_VEL
LIN {X 0,Y 378.917,Z 570.537,A -85,B 0,C 180,E1 -12346.015,E2 -12346.015} C_VEL
LIN {X 0,Y 379.815,Z 558.43,A -85,B 0,C 180,E1 -12346.944,E2 -12346.944} C_VEL
LIN {X 0,Y 380.543,Z 545.772,A -85,B 0,C 180,E1 -12347.672,E2 -12347.672} C_VEL
LIN {X 0,Y 381.146,Z 533.48,A -85,B 0,C 180,E1 -12348.164,E2 -12348.164} C_VEL
LIN {X 0,Y 381.478,Z 517.814,A -85,B 0,C 180,E1 -12348.53,E2 -12348.53} C_VEL
LIN {X 0,Y 382.211,Z 448.969,A -85,B 0,C 180,E1 -12349.828,E2 -12349.828} C_VEL
LIN {X 0,Y 377.937,Z 421.118,A -85,B 0,C 180,E1 -12350.592,E2 -12350.592} C_VEL
LIN {X 0,Y 378.419,Z 414.292,A -85,B 0,C 180,E1 -12352.091,E2 -12352.091} C_VEL
LIN {X 0,Y 378.823,Z 406.956,A -85,B 0,C 180,E1 -12353.798,E2 -12353.798} C_VEL
LIN {X 0,Y 376.517,Z 394.476,A -85,B 0,C 180,E1 -12356.913,E2 -12356.913} C_VEL
LIN {X 0,Y 376.06,Z 392.176,A -85,B 0,C 180,E1 -12357.589,E2 -12357.589} C_VEL
LIN {X 0,Y 375.958,Z 392.157,A -85,B 0,C 180,E1 -12361.561,E2 -12361.561} C_VEL
LIN {X 0,Y 375.958,Z 392.156,A -85,B 0,C 180,E1 -12365.415,E2 -12365.415} C_VEL
LIN {X 0,Y 375.976,Z 392.149,A -85,B 0,C 180,E1 -12368.27,E2 -12368.27} C_VEL
LIN {X 0,Y 375.935,Z 392.159,A -85,B 0,C 180,E1 -12371.6,E2 -12371.6} C_VEL
LIN {X 0,Y 375.978,Z 392.152,A -85,B 0,C 180,E1 -12375.26,E2 -12375.26} C_VEL
LIN {X 0,Y 375.988,Z 392.147,A -85,B 0,C 180,E1 -12378.389,E2 -12378.389} C_VEL
LIN {X 0,Y 375.966,Z 392.152,A -85,B 0,C 180,E1 -12381.911,E2 -12381.911} C_VEL
LIN {X 0,Y 375.977,Z 392.154,A -85,B 0,C 180,E1 -12385.332,E2 -12385.332} C_VEL
LIN {X 0,Y 375.954,Z 392.151,A -85,B 0,C 180,E1 -12388.437,E2 -12388.437} C_VEL
LIN {X 0,Y 375.992,Z 392.147,A -85,B 0,C 180,E1 -12392.141,E2 -12392.141} C_VEL
LIN {X 0,Y 376.001,Z 392.146,A -85,B 0,C 180,E1 -12394.538,E2 -12394.538} C_VEL
LIN {X 0,Y 375.954,Z 392.152,A -85,B 0,C 180,E1 -12398.045,E2 -12398.045} C_VEL
LIN {X 0,Y 376.019,Z 392.148,A -85,B 0,C 180,E1 -12401.474,E2 -12401.474} C_VEL
LIN {X 0,Y 376.053,Z 392.141,A -85,B 0,C 180,E1 -12404.832,E2 -12404.832} C_VEL
LIN {X 0,Y 376.044,Z 392.141,A -85,B 0,C 180,E1 -12408.136,E2 -12408.136} C_VEL
LIN {X 0,Y 376.214,Z 392.12,A -85,B 0,C 180,E1 -12411.918,E2 -12411.918} C_VEL
LIN {X 0,Y 376.166,Z 392.126,A -85,B 0,C 180,E1 -12414.64,E2 -12414.64} C_VEL
LIN {X 0,Y 376.348,Z 392.104,A -85,B 0,C 180,E1 -12417.859,E2 -12417.859} C_VEL
LIN {X 0,Y 376.483,Z 392.086,A -85,B 0,C 180,E1 -12420,E2 -12420} C_VEL
LIN {X 0,Y 376.185,Z 392.128,A -85,B 0,C 180,E1 -12423.213,E2 -12423.213} C_VEL
LIN {X 0,Y 376.222,Z 392.118,A -85,B 0,C 180,E1 -12426.629,E2 -12426.629} C_VEL
LIN {X 0,Y 376.114,Z 392.134,A -85,B 0,C 180,E1 -12429.682,E2 -12429.682} C_VEL
LIN {X 0,Y 376.084,Z 392.138,A -85,B 0,C 180,E1 -12433.658,E2 -12433.658} C_VEL
LIN {X 0,Y 376.038,Z 392.144,A -85,B 0,C 180,E1 -12437.607,E2 -12437.607} C_VEL
LIN {X 0,Y 375.974,Z 392.152,A -85,B 0,C 180,E1 -12440.832,E2 -12440.832} C_VEL
LIN {X 0,Y 375.989,Z 392.147,A -85,B 0,C 180,E1 -12444.282,E2 -12444.282} C_VEL
LIN {X 0,Y 376.015,Z 392.146,A -85,B 0,C 180,E1 -12446.652,E2 -12446.652} C_VEL
LIN {X 0,Y 375.973,Z 392.154,A -85,B 0,C 180,E1 -12449.079,E2 -12449.079} C_VEL
LIN {X 0,Y 375.946,Z 392.156,A -85,B 0,C 180,E1 -12452.829,E2 -12452.829} C_VEL
LIN {X 0,Y 375.955,Z 392.155,A -85,B 0,C 180,E1 -12455.416,E2 -12455.416} C_VEL
LIN {X 0,Y 375.972,Z 392.149,A -85,B 0,C 180,E1 -12458.271,E2 -12458.271} C_VEL
LIN {X 0,Y 375.932,Z 392.156,A -85,B 0,C 180,E1 -12461.601,E2 -12461.601} C_VEL
LIN {X 0,Y 375.951,Z 392.156,A -85,B 0,C 180,E1 -12465.265,E2 -12465.265} C_VEL
LIN {X 0,Y 375.979,Z 392.154,A -85,B 0,C 180,E1 -12469.139,E2 -12469.139} C_VEL
LIN {X 0,Y 375.967,Z 392.15,A -85,B 0,C 180,E1 -12471.912,E2 -12471.912} C_VEL
LIN {X 0,Y 375.979,Z 392.151,A -85,B 0,C 180,E1 -12475.333,E2 -12475.333} C_VEL
LIN {X 0,Y 375.957,Z 392.152,A -85,B 0,C 180,E1 -12478.438,E2 -12478.438} C_VEL
LIN {X 0,Y 375.983,Z 392.148,A -85,B 0,C 180,E1 -12482.141,E2 -12482.141} C_VEL
LIN {X 0,Y 376.007,Z 392.147,A -85,B 0,C 180,E1 -12484.539,E2 -12484.539} C_VEL
LIN {X 0,Y 375.964,Z 392.15,A -85,B 0,C 180,E1 -12488.046,E2 -12488.046} C_VEL
LIN {X 0,Y 376.01,Z 392.145,A -85,B 0,C 180,E1 -12491.473,E2 -12491.473} C_VEL
LIN {X 0,Y 376.06,Z 392.143,A -85,B 0,C 180,E1 -12494.833,E2 -12494.833} C_VEL
LIN {X 0,Y 376.119,Z 392.252,A -85,B 0,C 180,E1 -12497.523,E2 -12497.523} C_VEL
LIN {X 0,Y 378.243,Z 403.767,A -85,B 0,C 180,E1 -12500.643,E2 -12500.643} C_VEL
LIN {X 0,Y 378.134,Z 409.116,A -85,B 0,C 180,E1 -12501.987,E2 -12501.987} C_VEL
LIN {X 0,Y 377.818,Z 411.274,A -85,B 0,C 180,E1 -12502.451,E2 -12502.451} C_VEL
LIN {X 0,Y 379.131,Z 418.708,A -85,B 0,C 180,E1 -12502.696,E2 -12502.696} C_VEL
LIN {X 0,Y 382.541,Z 437.611,A -85,B 0,C 180,E1 -12503.219,E2 -12503.219} C_VEL
LIN {X 0,Y 381.281,Z 518.174,A -85,B 0,C 180,E1 -12504.745,E2 -12504.745} C_VEL
LIN {X 0,Y 380.845,Z 531.445,A -85,B 0,C 180,E1 -12505.206,E2 -12505.206} C_VEL
LIN {X 0,Y 380.162,Z 544.654,A -85,B 0,C 180,E1 -12505.892,E2 -12505.892} C_VEL
LIN {X 0,Y 379.434,Z 555.808,A -85,B 0,C 180,E1 -12506.682,E2 -12506.682} C_VEL
LIN {X 0,Y 378.454,Z 567.405,A -85,B 0,C 180,E1 -12507.738,E2 -12507.738} C_VEL
LIN {X 0,Y 377.659,Z 577.797,A -85,B 0,C 180,E1 -12508.933,E2 -12508.933} C_VEL
LIN {X 0,Y 376.813,Z 587.185,A -85,B 0,C 180,E1 -12510.267,E2 -12510.267} C_VEL
LIN {X 0,Y 375.962,Z 596.247,A -85,B 0,C 180,E1 -12511.874,E2 -12511.874} C_VEL
LIN {X 0,Y 375.421,Z 603.543,A -85,B 0,C 180,E1 -12513.488,E2 -12513.488} C_VEL
LIN {X 0,Y 374.997,Z 608.498,A -85,B 0,C 180,E1 -12514.838,E2 -12514.838} C_VEL
LIN {X 0,Y 374.822,Z 613.297,A -85,B 0,C 180,E1 -12516.459,E2 -12516.459} C_VEL
LIN {X 0,Y 374.57,Z 616.996,A -85,B 0,C 180,E1 -12518.089,E2 -12518.089} C_VEL
LIN {X 0,Y 374.38,Z 619.67,A -85,B 0,C 180,E1 -12519.726,E2 -12519.726} C_VEL
LIN {X 0,Y 374.36,Z 620.927,A -85,B 0,C 180,E1 -12520.82,E2 -12520.82} C_VEL
LIN {X 0,Y 374.404,Z 622.039,A -85,B 0,C 180,E1 -12522.551,E2 -12522.551} C_VEL
LIN {X 0,Y 374.269,Z 622.149,A -85,B 0,C 180,E1 -12524.129,E2 -12524.129} C_VEL
LIN {X 0,Y 374.307,Z 621.746,A -85,B 0,C 180,E1 -12525.239,E2 -12525.239} C_VEL
LIN {X 0,Y 374.442,Z 620.237,A -85,B 0,C 180,E1 -12526.95,E2 -12526.95} C_VEL
LIN {X 0,Y 373.891,Z 619.134,A -85,B 0,C 180,E1 -12527.833,E2 -12527.833} C_VEL
LIN {X 0,Y 371.259,Z 616.83,A -85,B 0,C 180,E1 -12529.264,E2 -12529.264} C_VEL
LIN {X 0,Y 369.089,Z 614.575,A -85,B 0,C 180,E1 -12530.399,E2 -12530.399} C_VEL
LIN {X 0,Y 368.287,Z 612.518,A -85,B 0,C 180,E1 -12531.254,E2 -12531.254} C_VEL
LIN {X 0,Y 368.293,Z 611.729,A -85,B 0,C 180,E1 -12531.537,E2 -12531.537} C_VEL
LIN {X 0,Y 368.91,Z 606.195,A -85,B 0,C 180,E1 -12533.284,E2 -12533.284} C_VEL
LIN {X 0,Y 369.805,Z 599.204,A -85,B 0,C 180,E1 -12535.014,E2 -12535.014} C_VEL
LIN {X 0,Y 370.725,Z 592.005,A -85,B 0,C 180,E1 -12536.454,E2 -12536.454} C_VEL
LIN {X 0,Y 371.837,Z 583.249,A -85,B 0,C 180,E1 -12537.89,E2 -12537.89} C_VEL
LIN {X 0,Y 372.968,Z 573.508,A -85,B 0,C 180,E1 -12539.18,E2 -12539.18} C_VEL
LIN {X 0,Y 374.203,Z 562.627,A -85,B 0,C 180,E1 -12540.332,E2 -12540.332} C_VEL
LIN {X 0,Y 375.264,Z 550.965,A -85,B 0,C 180,E1 -12541.311,E2 -12541.311} C_VEL
LIN {X 0,Y 376.257,Z 538.65,A -85,B 0,C 180,E1 -12542.084,E2 -12542.084} C_VEL
LIN {X 0,Y 377.051,Z 525.126,A -85,B 0,C 180,E1 -12542.68,E2 -12542.68} C_VEL
LIN {X 0,Y 377.499,Z 512.963,A -85,B 0,C 180,E1 -12543.013,E2 -12543.013} C_VEL
LIN {X 0,Y 378.773,Z 438.284,A -85,B 0,C 180,E1 -12544.467,E2 -12544.467} C_VEL
LIN {X 0,Y 374.093,Z 416.985,A -85,B 0,C 180,E1 -12545.25,E2 -12545.25} C_VEL
LIN {X 0,Y 372.686,Z 411.644,A -85,B 0,C 180,E1 -12545.499,E2 -12545.499} C_VEL
LIN {X 0,Y 372.031,Z 407.807,A -85,B 0,C 180,E1 -12546.516,E2 -12546.516} C_VEL
LIN {X 0,Y 369.885,Z 397.094,A -85,B 0,C 180,E1 -12549.69,E2 -12549.69} C_VEL
LIN {X 0,Y 368.953,Z 393.074,A -85,B 0,C 180,E1 -12551.007,E2 -12551.007} C_VEL
LIN {X 0,Y 368.986,Z 393.02,A -85,B 0,C 180,E1 -12554.806,E2 -12554.806} C_VEL
LIN {X 0,Y 368.936,Z 393.021,A -85,B 0,C 180,E1 -12558.185,E2 -12558.185} C_VEL
LIN {X 0,Y 368.907,Z 393.024,A -85,B 0,C 180,E1 -12561.358,E2 -12561.358} C_VEL
LIN {X 0,Y 368.931,Z 393.018,A -85,B 0,C 180,E1 -12565.146,E2 -12565.146} C_VEL
LIN {X 0,Y 368.922,Z 393.021,A -85,B 0,C 180,E1 -12569.046,E2 -12569.046} C_VEL
LIN {X 0,Y 368.98,Z 393.017,A -85,B 0,C 180,E1 -12571.564,E2 -12571.564} C_VEL
LIN {X 0,Y 368.95,Z 393.026,A -85,B 0,C 180,E1 -12575.224,E2 -12575.224} C_VEL
LIN {X 0,Y 368.963,Z 393.024,A -85,B 0,C 180,E1 -12578.959,E2 -12578.959} C_VEL
LIN {X 0,Y 368.984,Z 393.016,A -85,B 0,C 180,E1 -12582.257,E2 -12582.257} C_VEL
LIN {X 0,Y 369.029,Z 393.01,A -85,B 0,C 180,E1 -12586.227,E2 -12586.227} C_VEL
LIN {X 0,Y 369.064,Z 393.003,A -85,B 0,C 180,E1 -12590.132,E2 -12590.132} C_VEL
LIN {X 0,Y 369.18,Z 392.998,A -85,B 0,C 180,E1 -12592.342,E2 -12592.342} C_VEL
LIN {X 0,Y 369.138,Z 392.996,A -85,B 0,C 180,E1 -12594.538,E2 -12594.538} C_VEL
LIN {X 0,Y 369.317,Z 392.977,A -85,B 0,C 180,E1 -12597.819,E2 -12597.819} C_VEL
LIN {X 0,Y 369.452,Z 392.958,A -85,B 0,C 180,E1 -12600,E2 -12600} C_VEL
LIN {X 0,Y 369.311,Z 392.981,A -85,B 0,C 180,E1 -12602.181,E2 -12602.181} C_VEL
LIN {X 0,Y 369.201,Z 392.997,A -85,B 0,C 180,E1 -12606.558,E2 -12606.558} C_VEL
LIN {X 0,Y 369.131,Z 392.997,A -85,B 0,C 180,E1 -12608.761,E2 -12608.761} C_VEL
LIN {X 0,Y 369.005,Z 393.018,A -85,B 0,C 180,E1 -12612.093,E2 -12612.093} C_VEL
LIN {X 0,Y 368.99,Z 393.02,A -85,B 0,C 180,E1 -12615.465,E2 -12615.465} C_VEL
LIN {X 0,Y 368.976,Z 393.019,A -85,B 0,C 180,E1 -12618.893,E2 -12618.893} C_VEL
LIN {X 0,Y 368.926,Z 393.024,A -85,B 0,C 180,E1 -12622.396,E2 -12622.396} C_VEL
LIN {X 0,Y 368.993,Z 393.019,A -85,B 0,C 180,E1 -12625.981,E2 -12625.981} C_VEL
LIN {X 0,Y 368.955,Z 393.028,A -85,B 0,C 180,E1 -12628.812,E2 -12628.812} C_VEL
LIN {X 0,Y 368.892,Z 393.034,A -85,B 0,C 180,E1 -12632.239,E2 -12632.239} C_VEL
LIN {X 0,Y 368.924,Z 393.031,A -85,B 0,C 180,E1 -12635.002,E2 -12635.002} C_VEL
LIN {X 0,Y 368.909,Z 393.035,A -85,B 0,C 180,E1 -12638.642,E2 -12638.642} C_VEL
LIN {X 0,Y 368.937,Z 393.011,A -85,B 0,C 180,E1 -12642.021,E2 -12642.021} C_VEL
LIN {X 0,Y 368.921,Z 393.025,A -85,B 0,C 180,E1 -12645.184,E2 -12645.184} C_VEL
LIN {X 0,Y 368.888,Z 393.035,A -85,B 0,C 180,E1 -12648.18,E2 -12648.18} C_VEL
LIN {X 0,Y 368.908,Z 393.032,A -85,B 0,C 180,E1 -12651.36,E2 -12651.36} C_VEL
LIN {X 0,Y 368.935,Z 393.029,A -85,B 0,C 180,E1 -12655.147,E2 -12655.147} C_VEL
LIN {X 0,Y 368.928,Z 393.03,A -85,B 0,C 180,E1 -12659.047,E2 -12659.047} C_VEL
LIN {X 0,Y 368.941,Z 393.225,A -85,B 0,C 180,E1 -12660.077,E2 -12660.077} C_VEL
LIN {X 0,Y 371.275,Z 403.117,A -85,B 0,C 180,E1 -12662.981,E2 -12662.981} C_VEL
LIN {X 0,Y 373.039,Z 412.354,A -85,B 0,C 180,E1 -12665.515,E2 -12665.515} C_VEL
LIN {X 0,Y 372.973,Z 415.873,A -85,B 0,C 180,E1 -12666.397,E2 -12666.397} C_VEL
LIN {X 0,Y 372.522,Z 420.745,A -85,B 0,C 180,E1 -12667.524,E2 -12667.524} C_VEL
LIN {X 0,Y 375.5,Z 434.126,A -85,B 0,C 180,E1 -12668.063,E2 -12668.063} C_VEL
LIN {X 0,Y 378.632,Z 451.562,A -85,B 0,C 180,E1 -12668.648,E2 -12668.648} C_VEL
LIN {X 0,Y 377.244,Z 528.316,A -85,B 0,C 180,E1 -12670.16,E2 -12670.16} C_VEL
LIN {X 0,Y 376.6,Z 541.484,A -85,B 0,C 180,E1 -12670.621,E2 -12670.621} C_VEL
LIN {X 0,Y 375.674,Z 553.598,A -85,B 0,C 180,E1 -12671.245,E2 -12671.245} C_VEL
LIN {X 0,Y 374.6,Z 565.84,A -85,B 0,C 180,E1 -12672.109,E2 -12672.109} C_VEL
LIN {X 0,Y 373.359,Z 577.389,A -85,B 0,C 180,E1 -12673.178,E2 -12673.178} C_VEL
LIN {X 0,Y 372.101,Z 588.044,A -85,B 0,C 180,E1 -12674.42,E2 -12674.42} C_VEL
LIN {X 0,Y 371.091,Z 597.184,A -85,B 0,C 180,E1 -12675.748,E2 -12675.748} C_VEL
LIN {X 0,Y 370.077,Z 604.9,A -85,B 0,C 180,E1 -12677.107,E2 -12677.107} C_VEL
LIN {X 0,Y 369.185,Z 612.454,A -85,B 0,C 180,E1 -12678.749,E2 -12678.749} C_VEL
LIN {X 0,Y 368.345,Z 619.452,A -85,B 0,C 180,E1 -12680.667,E2 -12680.667} C_VEL
LIN {X 0,Y 367.855,Z 624.108,A -85,B 0,C 180,E1 -12682.315,E2 -12682.315} C_VEL
LIN {X 0,Y 367.571,Z 627.454,A -85,B 0,C 180,E1 -12683.852,E2 -12683.852} C_VEL
LIN {X 0,Y 367.469,Z 630.239,A -85,B 0,C 180,E1 -12685.613,E2 -12685.613} C_VEL
LIN {X 0,Y 367.356,Z 631.454,A -85,B 0,C 180,E1 -12686.71,E2 -12686.71} C_VEL
LIN {X 0,Y 367.317,Z 632.239,A -85,B 0,C 180,E1 -12687.807,E2 -12687.807} C_VEL
LIN {X 0,Y 367.351,Z 632.623,A -85,B 0,C 180,E1 -12688.904,E2 -12688.904} C_VEL
LIN {X 0,Y 367.389,Z 632.623,A -85,B 0,C 180,E1 -12690,E2 -12690} C_VEL
LIN {X 0,Y 367.352,Z 632.239,A -85,B 0,C 180,E1 -12691.096,E2 -12691.096} C_VEL
LIN {X 0,Y 367.319,Z 631.437,A -85,B 0,C 180,E1 -12692.193,E2 -12692.193} C_VEL
LIN {X 0,Y 367.353,Z 630.21,A -85,B 0,C 180,E1 -12693.29,E2 -12693.29} C_VEL
LIN {X 0,Y 367.45,Z 627.599,A -85,B 0,C 180,E1 -12694.938,E2 -12694.938} C_VEL
LIN {X 0,Y 367.566,Z 623.96,A -85,B 0,C 180,E1 -12696.588,E2 -12696.588} C_VEL
LIN {X 0,Y 367.896,Z 619.198,A -85,B 0,C 180,E1 -12698.237,E2 -12698.237} C_VEL
LIN {X 0,Y 368.415,Z 612.035,A -85,B 0,C 180,E1 -12700.163,E2 -12700.163} C_VEL
LIN {X 0,Y 369.078,Z 604.213,A -85,B 0,C 180,E1 -12701.812,E2 -12701.812} C_VEL
LIN {X 0,Y 369.829,Z 596.206,A -85,B 0,C 180,E1 -12703.182,E2 -12703.182} C_VEL
LIN {X 0,Y 370.685,Z 586.973,A -85,B 0,C 180,E1 -12704.478,E2 -12704.478} C_VEL
LIN {X 0,Y 371.499,Z 576.829,A -85,B 0,C 180,E1 -12705.639,E2 -12705.639} C_VEL
LIN {X 0,Y 372.4,Z 564.854,A -85,B 0,C 180,E1 -12706.726,E2 -12706.726} C_VEL
LIN {X 0,Y 373.311,Z 552.001,A -85,B 0,C 180,E1 -12707.601,E2 -12707.601} C_VEL
LIN {X 0,Y 374.03,Z 539.05,A -85,B 0,C 180,E1 -12708.238,E2 -12708.238} C_VEL
LIN {X 0,Y 374.464,Z 526.312,A -85,B 0,C 180,E1 -12708.64,E2 -12708.64} C_VEL
LIN {X 0,Y 375.42,Z 449.774,A -85,B 0,C 180,E1 -12710.118,E2 -12710.118} C_VEL
LIN {X 0,Y 370.991,Z 421.028,A -85,B 0,C 180,E1 -12710.927,E2 -12710.927} C_VEL
